C05442=1046.873,-51.756,-73.324,169.845,33.120,156.255
C05443=1046.866,-52.006,-73.312,169.843,33.118,156.255
C05444=1046.860,-52.255,-73.300,169.841,33.117,156.255
C05445=1046.854,-52.505,-73.288,169.839,33.117,156.255
C05446=1046.847,-52.754,-73.275,169.836,33.115,156.255
C05447=1046.841,-53.004,-73.262,169.834,33.114,156.255
C05448=1046.834,-53.254,-73.250,169.832,33.113,156.255
C05449=1046.828,-53.504,-73.238,169.830,33.112,156.255
C05450=1046.822,-53.753,-73.226,169.828,33.111,156.254
C05451=1046.815,-54.003,-73.214,169.826,33.110,156.254
C05452=1046.809,-54.253,-73.201,169.824,33.109,156.254
C05453=1046.802,-54.502,-73.189,169.822,33.108,156.254
C05454=1046.797,-54.752,-73.177,169.820,33.107,156.254
C05455=1046.790,-55.001,-73.165,169.817,33.106,156.254
C05456=1046.784,-55.251,-73.153,169.815,33.105,156.254
C05457=1046.778,-55.500,-73.140,169.813,33.104,156.254
C05458=1046.771,-55.749,-73.128,169.812,33.103,156.254
C05459=1046.764,-55.999,-73.116,169.810,33.102,156.253
C05460=1046.758,-56.249,-73.103,169.808,33.101,156.253
C05461=1046.752,-56.498,-73.092,169.806,33.100,156.253
C05462=1046.746,-56.748,-73.079,169.804,33.099,156.253
C05463=1046.739,-56.998,-73.067,169.801,33.098,156.253
C05464=1046.733,-57.247,-73.055,169.799,33.097,156.253
C05465=1046.727,-57.497,-73.043,169.797,33.096,156.253
C05466=1046.720,-57.747,-73.031,169.795,33.095,156.253
C05467=1046.714,-57.996,-73.019,169.793,33.094,156.253
C05468=1046.708,-58.246,-73.006,169.791,33.093,156.253
C05469=1046.701,-58.495,-72.994,169.789,33.092,156.253
C05470=1046.696,-58.746,-72.983,169.787,33.091,156.252
C05471=1046.689,-58.995,-72.971,169.784,33.090,156.252
C05472=1046.683,-59.245,-72.959,169.782,33.089,156.252
C05473=1046.677,-59.495,-72.946,169.780,33.088,156.252
C05474=1046.671,-59.744,-72.935,169.778,33.088,156.252
C05475=1046.664,-59.993,-72.923,169.776,33.086,156.252
C05476=1046.658,-60.243,-72.910,169.774,33.085,156.252
C05477=1046.651,-60.493,-72.898,169.772,33.085,156.252
C05478=1046.645,-60.742,-72.886,169.769,33.084,156.252
C05479=1046.639,-60.992,-72.874,169.767,33.082,156.252
C05480=1046.633,-61.242,-72.863,169.765,33.081,156.252
C05481=1046.626,-61.491,-72.851,169.763,33.081,156.251
C05482=1046.621,-61.741,-72.838,169.761,33.080,156.251
C05483=1046.614,-61.991,-72.826,169.759,33.079,156.251
C05484=1046.607,-62.240,-72.814,169.757,33.078,156.251
C05485=1046.602,-62.489,-72.802,169.755,33.077,156.251
C05486=1046.596,-62.740,-72.791,169.752,33.076,156.251
C05487=1046.589,-62.989,-72.779,169.750,33.075,156.251
C05488=1046.583,-63.239,-72.766,169.748,33.074,156.251
C05489=1046.576,-63.489,-72.754,169.746,33.073,156.251
C05490=1046.570,-63.737,-72.743,169.744,33.072,156.251
C05491=1046.565,-63.988,-72.731,169.742,33.071,156.251
C05492=1046.558,-64.238,-72.719,169.739,33.070,156.250
C05493=1046.551,-64.487,-72.707,169.738,33.069,156.250
C05494=1046.545,-64.736,-72.695,169.736,33.068,156.250
C05495=1046.540,-64.986,-72.684,169.734,33.067,156.250
C05496=1046.533,-65.236,-72.672,169.732,33.066,156.250
C05497=1046.527,-65.485,-72.660,169.730,33.065,156.250
C05498=1046.521,-65.735,-72.647,169.728,33.065,156.250
C05499=1046.515,-65.985,-72.636,169.725,33.064,156.250
C05500=1046.508,-66.235,-72.624,169.723,33.062,156.250
C05501=1046.503,-66.484,-72.612,169.721,33.061,156.250
C05502=1046.497,-66.734,-72.601,169.719,33.061,156.250
C05503=1046.489,-67.016,-72.587,169.716,33.060,156.250
C05504=1046.483,-67.299,-72.574,169.714,33.058,156.249
C05505=1046.476,-67.581,-72.560,169.712,33.057,156.249
C05506=1046.469,-67.863,-72.547,169.709,33.057,156.249
C05507=1046.462,-68.113,-72.535,169.707,33.056,156.249
C05508=1046.456,-68.362,-72.524,169.705,33.055,156.249
C05509=1046.450,-68.612,-72.513,169.703,33.054,156.249
C05510=1046.444,-68.862,-72.500,169.701,33.053,156.249
C05511=1046.438,-69.111,-72.489,169.698,33.052,156.249
C05512=1046.432,-69.361,-72.477,169.696,33.051,156.249
C05513=1046.425,-69.611,-72.465,169.694,33.050,156.249
C05514=1046.420,-69.860,-72.454,169.692,33.049,156.249
C05515=1046.413,-70.110,-72.442,169.690,33.049,156.248
C05516=1046.407,-70.360,-72.431,169.688,33.048,156.248
C05517=1046.401,-70.609,-72.419,169.685,33.047,156.248
C05518=1046.395,-70.859,-72.407,169.683,33.046,156.248
C05519=1046.389,-71.108,-72.396,169.681,33.045,156.248
C05520=1046.383,-71.358,-72.384,169.679,33.044,156.248
C05521=1046.376,-71.608,-72.372,169.677,33.043,156.248
C05522=1046.371,-71.857,-72.360,169.674,33.042,156.248
C05523=1046.365,-72.107,-72.349,169.672,33.041,156.248
C05524=1046.359,-72.356,-72.337,169.670,33.040,156.248
C05525=1046.352,-72.607,-72.326,169.669,33.040,156.248
C05526=1046.347,-72.856,-72.314,169.667,33.039,156.248
C05527=1046.341,-73.106,-72.303,169.665,33.038,156.248
C05528=1046.334,-73.356,-72.291,169.662,33.037,156.248
C05529=1046.328,-73.605,-72.280,169.660,33.036,156.247
C05530=1046.322,-73.855,-72.269,169.658,33.035,156.247
C05531=1046.317,-74.104,-72.256,169.656,33.035,156.247
C05532=1046.310,-74.355,-72.245,169.654,33.034,156.247
C05533=1046.304,-74.603,-72.234,169.651,33.033,156.247
C05534=1046.298,-74.854,-72.222,169.649,33.032,156.247
C05535=1046.292,-75.104,-72.211,169.647,33.031,156.247
C05536=1046.285,-75.352,-72.200,169.645,33.030,156.247
C05537=1046.278,-75.603,-72.189,169.643,33.030,156.247
C05538=1046.273,-75.852,-72.178,169.640,33.029,156.247
C05539=1046.266,-76.102,-72.166,169.638,33.028,156.247
C05540=1046.260,-76.351,-72.155,169.636,33.028,156.247
C05541=1046.254,-76.601,-72.144,169.634,33.027,156.247
C05542=1046.248,-76.850,-72.132,169.632,33.026,156.247
C05543=1046.242,-77.100,-72.121,169.629,33.025,156.247
C05544=1046.235,-77.351,-72.110,169.627,33.024,156.247
C05545=1046.229,-77.599,-72.098,169.625,33.024,156.247
C05546=1046.223,-77.850,-72.087,169.623,33.023,156.247
C05547=1046.217,-78.099,-72.076,169.620,33.022,156.247
C05548=1046.210,-78.349,-72.064,169.618,33.021,156.246
C05549=1046.205,-78.598,-72.053,169.616,33.021,156.246
C05550=1046.198,-78.848,-72.042,169.614,33.020,156.246
C05551=1046.193,-79.098,-72.031,169.612,33.020,156.246
C05552=1046.186,-79.348,-72.020,169.609,33.019,156.246
C05553=1046.180,-79.597,-72.008,169.607,33.018,156.246
C05554=1046.174,-79.847,-71.997,169.605,33.017,156.246
C05555=1046.167,-80.096,-71.987,169.603,33.016,156.246
C05556=1046.161,-80.346,-71.975,169.601,33.016,156.246
C05557=1046.155,-80.596,-71.965,169.599,33.015,156.246
C05558=1046.149,-80.846,-71.953,169.597,33.014,156.246
C05559=1046.142,-81.095,-71.942,169.595,33.014,156.246
C05560=1046.136,-81.345,-71.931,169.592,33.013,156.246
C05561=1046.130,-81.594,-71.920,169.590,33.012,156.246
C05562=1046.124,-81.845,-71.909,169.588,33.012,156.246
C05563=1046.117,-82.094,-71.899,169.586,33.011,156.246
C05564=1046.111,-82.344,-71.887,169.583,33.011,156.246
C05565=1046.105,-82.593,-71.877,169.581,33.010,156.246
C05566=1046.098,-82.843,-71.866,169.579,33.009,156.246
C05567=1046.091,-83.127,-71.853,169.576,33.009,156.246
C05568=1046.084,-83.412,-71.840,169.574,33.008,156.246
C05569=1046.077,-83.697,-71.828,169.571,33.007,156.246
C05570=1046.070,-83.981,-71.816,169.569,33.007,156.246
C05571=1046.063,-84.231,-71.804,169.566,33.006,156.246
C05572=1046.058,-84.480,-71.794,169.564,33.006,156.246
C05573=1046.051,-84.730,-71.783,169.562,33.005,156.246
C05574=1046.045,-84.980,-71.772,169.560,33.005,156.246
C05575=1046.039,-85.229,-71.761,169.557,33.004,156.246
C05576=1046.032,-85.479,-71.751,169.555,33.003,156.246
C05577=1046.026,-85.729,-71.740,169.553,33.003,156.246
C05578=1046.020,-85.979,-71.728,169.551,33.002,156.246
C05579=1046.013,-86.228,-71.718,169.548,33.002,156.246
C05580=1046.008,-86.477,-71.707,169.546,33.001,156.246
C05581=1046.001,-86.728,-71.696,169.544,33.000,156.246
C05582=1045.995,-86.977,-71.686,169.542,33.000,156.246
C05583=1045.989,-87.227,-71.674,169.540,32.999,156.246
C05584=1045.983,-87.477,-71.664,169.538,32.999,156.245
C05585=1045.977,-87.726,-71.654,169.536,32.998,156.246
C05586=1045.970,-87.977,-71.643,169.533,32.997,156.245
C05587=1045.965,-88.226,-71.632,169.531,32.997,156.246
C05588=1045.958,-88.475,-71.622,169.529,32.996,156.245
C05589=1045.952,-88.725,-71.610,169.527,32.996,156.246
C05590=1045.946,-88.975,-71.600,169.524,32.995,156.245
C05591=1045.940,-89.224,-71.589,169.522,32.995,156.245
C05592=1045.933,-89.474,-71.578,169.520,32.994,156.245
C05593=1045.927,-89.724,-71.567,169.518,32.994,156.245
C05594=1045.921,-89.974,-71.558,169.515,32.993,156.245
C05595=1045.915,-90.224,-71.546,169.513,32.993,156.245
C05596=1045.909,-90.473,-71.535,169.511,32.992,156.245
C05597=1045.903,-90.722,-71.525,169.508,32.992,156.245
C05598=1045.896,-90.973,-71.514,169.506,32.991,156.245
C05599=1045.890,-91.222,-71.504,169.504,32.991,156.245
C05600=1045.884,-91.472,-71.493,169.502,32.990,156.245
C05601=1045.878,-91.722,-71.482,169.499,32.990,156.245
C05602=1045.872,-91.971,-71.472,169.497,32.989,156.245
C05603=1045.866,-92.221,-71.461,169.495,32.989,156.245
C05604=1045.860,-92.470,-71.450,169.493,32.988,156.245
C05605=1045.853,-92.721,-71.440,169.490,32.988,156.245
C05606=1045.848,-92.970,-71.429,169.488,32.987,156.245
C05607=1045.841,-93.219,-71.419,169.486,32.987,156.245
C05608=1045.835,-93.469,-71.408,169.483,32.986,156.245
C05609=1045.829,-93.720,-71.398,169.481,32.986,156.245
C05610=1045.823,-93.969,-71.387,169.479,32.985,156.245
C05611=1045.817,-94.218,-71.377,169.477,32.985,156.245
C05612=1045.811,-94.468,-71.367,169.475,32.984,156.245
C05613=1045.805,-94.718,-71.356,169.473,32.983,156.245
C05614=1045.799,-94.968,-71.345,169.471,32.983,156.245
C05615=1045.792,-95.217,-71.335,169.468,32.982,156.245
C05616=1045.787,-95.467,-71.324,169.466,32.982,156.245
C05617=1045.781,-95.716,-71.314,169.464,32.982,156.245
C05618=1045.775,-95.966,-71.303,169.462,32.981,156.245
C05619=1045.769,-96.217,-71.293,169.459,32.981,156.245
C05620=1045.762,-96.466,-71.282,169.457,32.980,156.245
C05621=1045.757,-96.716,-71.272,169.455,32.980,156.245
C05622=1045.750,-96.965,-71.262,169.452,32.980,156.245
C05623=1045.745,-97.215,-71.251,169.450,32.979,156.245
C05624=1045.738,-97.465,-71.241,169.448,32.979,156.245
C05625=1045.732,-97.715,-71.230,169.446,32.978,156.245
C05626=1045.726,-97.964,-71.221,169.443,32.977,156.245
C05627=1045.720,-98.214,-71.210,169.441,32.977,156.245
C05628=1045.714,-98.463,-71.200,169.439,32.977,156.246
C05629=1045.707,-98.714,-71.190,169.436,32.977,156.246
C05630=1045.701,-98.963,-71.179,169.434,32.977,156.246
C05631=1045.695,-99.250,-71.168,169.431,32.976,156.246
C05632=1045.687,-99.536,-71.156,169.429,32.975,156.246
C05633=1045.680,-99.824,-71.145,169.426,32.975,156.246
C05634=1045.673,-100.111,-71.132,169.423,32.975,156.246
C05635=1045.667,-100.360,-71.123,169.421,32.974,156.246
C05636=1045.660,-100.610,-71.112,169.419,32.974,156.246
C05637=1045.655,-100.860,-71.102,169.416,32.974,156.246
C05638=1045.648,-101.109,-71.092,169.415,32.973,156.246
C05639=1045.642,-101.359,-71.082,169.413,32.973,156.246
C05640=1045.636,-101.608,-71.071,169.410,32.973,156.246
C05641=1045.629,-101.859,-71.061,169.408,32.972,156.246
C05642=1045.623,-102.108,-71.051,169.406,32.972,156.246
C05643=1045.618,-102.358,-71.041,169.403,32.972,156.246
C05644=1045.611,-102.608,-71.031,169.401,32.971,156.246
C05645=1045.605,-102.857,-71.021,169.399,32.971,156.246
C05646=1045.600,-103.107,-71.011,169.397,32.971,156.246
C05647=1045.593,-103.356,-71.001,169.394,32.971,156.246
C05648=1045.587,-103.606,-70.991,169.392,32.970,156.246
C05649=1045.581,-103.856,-70.982,169.390,32.970,156.246
C05650=1045.575,-104.105,-70.971,169.387,32.969,156.246
C05651=1045.569,-104.355,-70.961,169.385,32.969,156.246
C05652=1045.562,-104.606,-70.951,169.383,32.969,156.246
C05653=1045.556,-104.855,-70.940,169.380,32.969,156.246
C05654=1045.550,-105.105,-70.931,169.378,32.969,156.246
C05655=1045.544,-105.355,-70.921,169.376,32.968,156.246
C05656=1045.537,-105.604,-70.911,169.373,32.968,156.246
C05657=1045.532,-105.854,-70.901,169.371,32.968,156.247
C05658=1045.526,-106.104,-70.891,169.369,32.968,156.247
C05659=1045.520,-106.354,-70.882,169.366,32.967,156.247
C05660=1045.513,-106.603,-70.871,169.364,32.967,156.247
C05661=1045.507,-106.853,-70.862,169.362,32.966,156.247
C05662=1045.502,-107.103,-70.852,169.359,32.966,156.247
C05663=1045.495,-107.352,-70.842,169.357,32.966,156.247
C05664=1045.489,-107.602,-70.832,169.355,32.966,156.247
C05665=1045.483,-107.851,-70.822,169.353,32.966,156.247
C05666=1045.477,-108.101,-70.813,169.351,32.965,156.247
C05667=1045.470,-108.351,-70.803,169.349,32.966,156.247
C05668=1045.465,-108.601,-70.792,169.346,32.965,156.247
C05669=1045.459,-108.850,-70.783,169.344,32.965,156.247
C05670=1045.452,-109.100,-70.773,169.341,32.965,156.247
C05671=1045.446,-109.350,-70.763,169.339,32.965,156.247
C05672=1045.440,-109.600,-70.754,169.337,32.965,156.247
C05673=1045.434,-109.850,-70.744,169.334,32.964,156.247
C05674=1045.427,-110.099,-70.734,169.332,32.964,156.247
C05675=1045.421,-110.348,-70.725,169.330,32.964,156.247
C05676=1045.415,-110.598,-70.715,169.327,32.964,156.247
C05677=1045.409,-110.848,-70.705,169.325,32.963,156.248
C05678=1045.403,-111.098,-70.695,169.323,32.964,156.248
C05679=1045.397,-111.348,-70.686,169.320,32.964,156.248
C05680=1045.391,-111.598,-70.676,169.318,32.963,156.248
C05681=1045.385,-111.848,-70.667,169.316,32.963,156.248
C05682=1045.379,-112.097,-70.657,169.313,32.963,156.248
C05683=1045.373,-112.347,-70.647,169.311,32.963,156.248
C05684=1045.366,-112.597,-70.638,169.308,32.962,156.248
C05685=1045.360,-112.846,-70.628,169.306,32.962,156.248
C05686=1045.354,-113.096,-70.618,169.304,32.963,156.248
C05687=1045.348,-113.346,-70.608,169.301,32.962,156.248
C05688=1045.342,-113.595,-70.599,169.299,32.962,156.248
C05689=1045.336,-113.845,-70.590,169.297,32.962,156.248
C05690=1045.330,-114.094,-70.580,169.295,32.962,156.248
C05691=1045.323,-114.344,-70.570,169.293,32.962,156.248
C05692=1045.317,-114.594,-70.561,169.291,32.962,156.249
C05693=1045.311,-114.844,-70.551,169.288,32.962,156.249
C05694=1045.305,-115.094,-70.542,169.286,32.962,156.249
C05695=1045.298,-115.380,-70.531,169.283,32.961,156.249
C05696=1045.291,-115.665,-70.520,169.280,32.962,156.249
C05697=1045.284,-115.952,-70.509,169.278,32.961,156.249
C05698=1045.277,-116.237,-70.499,169.275,32.961,156.249
C05699=1045.271,-116.487,-70.489,169.273,32.962,156.249
C05700=1045.265,-116.736,-70.480,169.270,32.961,156.249
C05701=1045.259,-116.986,-70.470,169.268,32.961,156.249
C05702=1045.253,-117.237,-70.461,169.266,32.962,156.249
C05703=1045.247,-117.486,-70.452,169.263,32.961,156.250
C05704=1045.240,-117.736,-70.442,169.261,32.961,156.250
C05705=1045.235,-117.985,-70.433,169.258,32.961,156.250
C05706=1045.229,-118.235,-70.423,169.256,32.961,156.250
C05707=1045.223,-118.485,-70.414,169.254,32.961,156.250
C05708=1045.216,-118.734,-70.405,169.251,32.961,156.250
C05709=1045.210,-118.985,-70.396,169.249,32.961,156.250
C05710=1045.204,-119.235,-70.386,169.247,32.961,156.250
C05711=1045.198,-119.484,-70.377,169.244,32.961,156.250
C05712=1045.192,-119.733,-70.368,169.242,32.961,156.250
C05713=1045.186,-119.983,-70.358,169.239,32.961,156.250
C05714=1045.180,-120.234,-70.349,169.237,32.961,156.251
C05715=1045.174,-120.483,-70.340,169.235,32.961,156.251
C05716=1045.167,-120.732,-70.331,169.233,32.961,156.251
C05717=1045.161,-120.982,-70.321,169.231,32.961,156.251
C05718=1045.155,-121.232,-70.312,169.228,32.961,156.251
C05719=1045.149,-121.482,-70.303,169.226,32.962,156.251
C05720=1045.143,-121.732,-70.293,169.224,32.961,156.251
C05721=1045.137,-121.981,-70.284,169.221,32.962,156.251
C05722=1045.130,-122.231,-70.275,169.219,32.961,156.251
C05723=1045.125,-122.481,-70.266,169.217,32.961,156.251
C05724=1045.118,-122.731,-70.257,169.214,32.962,156.251
C05725=1045.113,-122.980,-70.248,169.212,32.961,156.252
C05726=1045.107,-123.230,-70.239,169.209,32.962,156.252
C05727=1045.101,-123.480,-70.229,169.207,32.962,156.252
C05728=1045.094,-123.730,-70.220,169.205,32.962,156.252
C05729=1045.089,-123.979,-70.212,169.202,32.962,156.252
C05730=1045.083,-124.229,-70.202,169.200,32.962,156.252
C05731=1045.076,-124.479,-70.193,169.197,32.962,156.252
C05732=1045.070,-124.729,-70.184,169.195,32.962,156.252
C05733=1045.064,-124.978,-70.175,169.193,32.962,156.252
C05734=1045.058,-125.228,-70.166,169.190,32.963,156.253
C05735=1045.052,-125.478,-70.157,169.188,32.962,156.253
C05736=1045.045,-125.728,-70.148,169.185,32.963,156.253
C05737=1045.040,-125.978,-70.139,169.183,32.963,156.253
C05738=1045.034,-126.227,-70.130,169.181,32.963,156.253
C05739=1045.027,-126.478,-70.122,169.178,32.963,156.253
C05740=1045.022,-126.727,-70.112,169.176,32.963,156.253
C05741=1045.015,-126.976,-70.103,169.174,32.964,156.253
C05742=1045.009,-127.227,-70.094,169.172,32.964,156.254
C05743=1045.003,-127.476,-70.085,169.170,32.964,156.254
C05744=1044.997,-127.726,-70.076,169.167,32.964,156.254
C05745=1044.992,-127.975,-70.067,169.165,32.964,156.254
C05746=1044.986,-128.225,-70.057,169.163,32.963,156.254
C05747=1044.982,-128.475,-70.047,169.161,32.962,156.254
C05748=1044.980,-128.725,-70.035,169.159,32.961,156.253
C05749=1044.978,-128.975,-70.024,169.157,32.959,156.253
C05750=1044.977,-129.225,-70.011,169.155,32.957,156.253
C05751=1044.977,-129.475,-69.999,169.153,32.954,156.252
C05752=1044.978,-129.725,-69.985,169.152,32.951,156.252
C05753=1044.979,-129.976,-69.971,169.150,32.947,156.251
C05754=1044.982,-130.225,-69.957,169.149,32.943,156.251
C05755=1044.986,-130.476,-69.941,169.148,32.938,156.250
C05756=1044.990,-130.727,-69.925,169.147,32.933,156.249
C05757=1044.995,-130.977,-69.908,169.146,32.927,156.248
C05758=1045.002,-131.227,-69.891,169.145,32.921,156.247
C05759=1044.646,-131.251,-70.134,169.099,33.102,156.280
C05760=1044.641,-131.000,-70.151,169.100,33.108,156.281
C05761=1044.635,-130.751,-70.168,169.101,33.114,156.282
C05762=1044.631,-130.500,-70.184,169.102,33.119,156.283
C05763=1044.627,-130.249,-70.199,169.103,33.124,156.283
C05764=1044.624,-129.999,-70.214,169.104,33.128,156.284
C05765=1044.622,-129.749,-70.229,169.105,33.131,156.285
C05766=1044.622,-129.499,-70.242,169.107,33.135,156.285
C05767=1044.622,-129.248,-70.255,169.108,33.138,156.285
C05768=1044.623,-128.998,-70.268,169.110,33.140,156.286
C05769=1044.625,-128.749,-70.279,169.112,33.142,156.286
C05770=1044.627,-128.498,-70.291,169.114,33.144,156.286
C05771=1044.631,-128.249,-70.301,169.116,33.145,156.286
C05772=1044.636,-127.999,-70.311,169.118,33.145,156.286
C05773=1044.641,-127.749,-70.320,169.121,33.145,156.286
C05774=1044.648,-127.500,-70.329,169.123,33.145,156.286
C05775=1044.653,-127.251,-70.338,169.125,33.145,156.286
C05776=1044.659,-127.000,-70.347,169.128,33.144,156.286
C05777=1044.666,-126.751,-70.356,169.130,33.145,156.286
C05778=1044.671,-126.501,-70.364,169.133,33.144,156.286
C05779=1044.677,-126.251,-70.374,169.135,33.144,156.286
C05780=1044.684,-126.001,-70.382,169.138,33.144,156.285
C05781=1044.690,-125.751,-70.392,169.140,33.144,156.285
C05782=1044.696,-125.502,-70.400,169.142,33.144,156.285
C05783=1044.702,-125.252,-70.409,169.145,33.143,156.285
C05784=1044.709,-125.002,-70.419,169.147,33.143,156.285
C05785=1044.714,-124.753,-70.427,169.149,33.143,156.285
C05786=1044.721,-124.503,-70.436,169.151,33.143,156.285
C05787=1044.727,-124.253,-70.446,169.153,33.143,156.285
C05788=1044.733,-124.003,-70.455,169.156,33.143,156.285
C05789=1044.738,-123.754,-70.464,169.158,33.143,156.285
C05790=1044.745,-123.504,-70.473,169.161,33.142,156.284
C05791=1044.751,-123.254,-70.482,169.163,33.143,156.284
C05792=1044.757,-123.004,-70.491,169.165,33.142,156.284
C05793=1044.763,-122.755,-70.500,169.168,33.142,156.284
C05794=1044.769,-122.505,-70.509,169.170,33.142,156.284
C05795=1044.775,-122.255,-70.519,169.173,33.142,156.284
C05796=1044.782,-122.005,-70.528,169.175,33.142,156.284
C05797=1044.787,-121.756,-70.536,169.177,33.142,156.284
C05798=1044.793,-121.506,-70.546,169.180,33.142,156.284
C05799=1044.799,-121.256,-70.555,169.182,33.142,156.283
C05800=1044.806,-121.006,-70.565,169.185,33.142,156.283
C05801=1044.812,-120.756,-70.574,169.187,33.142,156.283
C05802=1044.817,-120.507,-70.583,169.189,33.142,156.283
C05803=1044.824,-120.257,-70.592,169.192,33.141,156.283
C05804=1044.830,-120.008,-70.602,169.194,33.142,156.283
C05805=1044.836,-119.758,-70.611,169.197,33.141,156.283
C05806=1044.842,-119.507,-70.620,169.199,33.141,156.283
C05807=1044.848,-119.258,-70.629,169.201,33.142,156.283
C05808=1044.854,-119.008,-70.639,169.204,33.141,156.283
C05809=1044.860,-118.759,-70.648,169.206,33.141,156.283
C05810=1044.866,-118.509,-70.658,169.208,33.142,156.282
C05811=1044.873,-118.259,-70.667,169.210,33.141,156.282
C05812=1044.879,-118.009,-70.676,169.212,33.141,156.282
C05813=1044.885,-117.760,-70.685,169.215,33.141,156.282
C05814=1044.891,-117.510,-70.694,169.217,33.141,156.282
C05815=1044.897,-117.260,-70.704,169.220,33.141,156.282
C05816=1044.903,-117.010,-70.714,169.222,33.141,156.282
C05817=1044.909,-116.761,-70.723,169.224,33.141,156.282
C05818=1044.915,-116.511,-70.733,169.227,33.141,156.282
C05819=1044.922,-116.261,-70.742,169.229,33.141,156.282
C05820=1044.929,-115.975,-70.752,169.232,33.141,156.282
C05821=1044.936,-115.689,-70.764,169.235,33.141,156.281
C05822=1044.943,-115.403,-70.774,169.237,33.141,156.281
C05823=1044.949,-115.118,-70.785,169.240,33.141,156.281
C05824=1044.956,-114.868,-70.795,169.242,33.141,156.281
C05825=1044.962,-114.618,-70.804,169.245,33.142,156.281
C05826=1044.968,-114.369,-70.814,169.247,33.141,156.281
C05827=1044.974,-114.119,-70.824,169.249,33.141,156.281
C05828=1044.980,-113.869,-70.833,169.252,33.142,156.281
C05829=1044.986,-113.619,-70.843,169.254,33.142,156.281
C05830=1044.992,-113.370,-70.852,169.257,33.142,156.281
C05831=1044.998,-113.120,-70.861,169.259,33.142,156.281
C05832=1045.004,-112.870,-70.871,169.261,33.142,156.281
C05833=1045.011,-112.621,-70.881,169.264,33.142,156.281
C05834=1045.017,-112.371,-70.890,169.266,33.142,156.281
C05835=1045.023,-112.121,-70.900,169.268,33.143,156.280
C05836=1045.029,-111.871,-70.909,169.270,33.142,156.280
C05837=1045.035,-111.621,-70.919,169.272,33.142,156.280
C05838=1045.041,-111.371,-70.929,169.275,33.143,156.280
C05839=1045.047,-111.122,-70.939,169.277,33.143,156.280
C05840=1045.053,-110.872,-70.948,169.279,33.143,156.280
C05841=1045.059,-110.622,-70.958,169.282,33.143,156.280
C05842=1045.066,-110.373,-70.968,169.284,33.143,156.280
C05843=1045.072,-110.123,-70.978,169.286,33.143,156.280
C05844=1045.078,-109.873,-70.987,169.289,33.143,156.280
C05845=1045.084,-109.623,-70.997,169.291,33.143,156.280
C05846=1045.090,-109.374,-71.006,169.293,33.144,156.280
C05847=1045.096,-109.124,-71.016,169.296,33.144,156.280
C05848=1045.103,-108.874,-71.025,169.298,33.144,156.280
C05849=1045.108,-108.624,-71.036,169.301,33.144,156.280
C05850=1045.115,-108.375,-71.046,169.303,33.145,156.280
C05851=1045.121,-108.125,-71.055,169.305,33.145,156.280
C05852=1045.127,-107.875,-71.065,169.308,33.144,156.279
C05853=1045.133,-107.625,-71.075,169.310,33.144,156.279
C05854=1045.140,-107.376,-71.085,169.312,33.145,156.279
C05855=1045.146,-107.126,-71.094,169.315,33.145,156.279
C05856=1045.151,-106.876,-71.105,169.317,33.145,156.279
C05857=1045.157,-106.626,-71.114,169.319,33.145,156.279
C05858=1045.164,-106.377,-71.124,169.322,33.146,156.279
C05859=1045.170,-106.127,-71.134,169.324,33.146,156.279
C05860=1045.175,-105.877,-71.144,169.326,33.146,156.279
C05861=1045.182,-105.628,-71.154,169.329,33.146,156.279
C05862=1045.188,-105.378,-71.164,169.331,33.146,156.279
C05863=1045.194,-105.129,-71.174,169.333,33.147,156.279
C05864=1045.200,-104.878,-71.184,169.335,33.147,156.279
C05865=1045.206,-104.629,-71.194,169.337,33.148,156.279
C05866=1045.212,-104.379,-71.204,169.339,33.148,156.279
C05867=1045.219,-104.129,-71.213,169.342,33.148,156.279
C05868=1045.225,-103.879,-71.224,169.344,33.148,156.279
C05869=1045.231,-103.630,-71.234,169.346,33.148,156.279
C05870=1045.237,-103.380,-71.244,169.349,33.149,156.279
C05871=1045.243,-103.130,-71.254,169.351,33.149,156.279
C05872=1045.249,-102.881,-71.264,169.353,33.149,156.279
C05873=1045.256,-102.631,-71.274,169.356,33.149,156.278
C05874=1045.262,-102.382,-71.284,169.358,33.150,156.278
C05875=1045.267,-102.132,-71.295,169.360,33.150,156.278
C05876=1045.274,-101.882,-71.304,169.363,33.151,156.278
C05877=1045.280,-101.632,-71.314,169.365,33.151,156.278
C05878=1045.286,-101.382,-71.325,169.367,33.151,156.278
C05879=1045.292,-101.133,-71.335,169.370,33.151,156.278
C05880=1045.299,-100.883,-71.345,169.372,33.151,156.278
C05881=1045.304,-100.633,-71.355,169.374,33.152,156.278
C05882=1045.311,-100.384,-71.365,169.377,33.152,156.278
C05883=1045.317,-100.134,-71.375,169.379,33.153,156.278
C05884=1045.324,-99.847,-71.387,169.382,33.153,156.278
C05885=1045.331,-99.560,-71.399,169.384,33.153,156.278
C05886=1045.339,-99.273,-71.411,169.387,33.153,156.278
C05887=1045.345,-98.986,-71.422,169.390,33.154,156.278
C05888=1045.351,-98.737,-71.432,169.392,33.155,156.278
C05889=1045.358,-98.487,-71.442,169.394,33.155,156.278
C05890=1045.364,-98.237,-71.453,169.397,33.155,156.278
C05891=1045.370,-97.987,-71.463,169.399,33.155,156.278
C05892=1045.376,-97.738,-71.473,169.400,33.155,156.278
C05893=1045.382,-97.489,-71.484,169.403,33.156,156.278
C05894=1045.389,-97.238,-71.494,169.405,33.156,156.278
C05895=1045.395,-96.989,-71.505,169.407,33.157,156.278
C05896=1045.401,-96.739,-71.514,169.410,33.158,156.278
C05897=1045.406,-96.489,-71.525,169.412,33.158,156.278
C05898=1045.412,-96.240,-71.536,169.414,33.158,156.278
C05899=1045.418,-95.990,-71.546,169.417,33.159,156.278
C05900=1045.425,-95.740,-71.557,169.419,33.159,156.278
C05901=1045.431,-95.491,-71.567,169.421,33.159,156.278
C05902=1045.437,-95.241,-71.577,169.423,33.160,156.278
C05903=1045.443,-94.991,-71.588,169.426,33.160,156.278
C05904=1045.449,-94.742,-71.598,169.428,33.161,156.278
C05905=1045.455,-94.491,-71.609,169.430,33.161,156.278
C05906=1045.461,-94.242,-71.619,169.433,33.161,156.278
C05907=1045.467,-93.992,-71.630,169.435,33.162,156.278
C05908=1045.474,-93.743,-71.640,169.437,33.162,156.278
C05909=1045.480,-93.493,-71.651,169.439,33.163,156.278
C05910=1045.485,-93.243,-71.662,169.442,33.164,156.278
C05911=1045.492,-92.994,-71.672,169.444,33.164,156.278
C05912=1045.498,-92.744,-71.683,169.446,33.165,156.278
C05913=1045.504,-92.494,-71.693,169.449,33.165,156.278
C05914=1045.510,-92.244,-71.704,169.451,33.166,156.278
C05915=1045.516,-91.995,-71.715,169.453,33.166,156.278
C05916=1045.522,-91.746,-71.725,169.456,33.167,156.278
C05917=1045.528,-91.495,-71.736,169.458,33.167,156.278
C05918=1045.534,-91.245,-71.746,169.460,33.167,156.278
C05919=1045.541,-90.996,-71.757,169.462,33.168,156.278
C05920=1045.547,-90.746,-71.768,169.465,33.168,156.278
C05921=1045.553,-90.497,-71.778,169.467,33.169,156.278
C05922=1045.559,-90.247,-71.789,169.468,33.169,156.278
C05923=1045.565,-89.997,-71.799,169.470,33.170,156.278
C05924=1045.572,-89.747,-71.810,169.473,33.170,156.278
C05925=1045.577,-89.498,-71.821,169.475,33.171,156.278
C05926=1045.583,-89.248,-71.832,169.477,33.171,156.278
C05927=1045.590,-88.999,-71.842,169.480,33.172,156.278
C05928=1045.596,-88.749,-71.853,169.482,33.172,156.278
C05929=1045.602,-88.500,-71.864,169.484,33.173,156.278
C05930=1045.609,-88.250,-71.875,169.486,33.173,156.278
C05931=1045.614,-88.000,-71.885,169.489,33.174,156.278
C05932=1045.621,-87.749,-71.896,169.491,33.174,156.278
C05933=1045.627,-87.500,-71.906,169.493,33.175,156.278
C05934=1045.633,-87.251,-71.917,169.496,33.175,156.278
C05935=1045.639,-87.000,-71.928,169.498,33.176,156.278
C05936=1045.646,-86.751,-71.939,169.500,33.176,156.278
C05937=1045.651,-86.502,-71.950,169.502,33.177,156.278
C05938=1045.658,-86.252,-71.961,169.505,33.178,156.278
C05939=1045.664,-86.002,-71.971,169.507,33.178,156.278
C05940=1045.670,-85.752,-71.982,169.509,33.179,156.278
C05941=1045.676,-85.503,-71.993,169.511,33.179,156.278
C05942=1045.683,-85.254,-72.004,169.514,33.180,156.278
C05943=1045.689,-85.003,-72.015,169.516,33.180,156.278
C05944=1045.695,-84.754,-72.026,169.518,33.181,156.278
C05945=1045.702,-84.504,-72.036,169.521,33.182,156.278
C05946=1045.708,-84.255,-72.047,169.523,33.182,156.278
C05947=1045.714,-84.004,-72.058,169.525,33.183,156.278
C05948=1045.721,-83.720,-72.071,169.528,33.183,156.278
C05949=1045.728,-83.436,-72.083,169.530,33.184,156.278
C05950=1045.735,-83.151,-72.096,169.533,33.185,156.278
C05951=1045.742,-82.866,-72.108,169.535,33.185,156.278
C05952=1045.749,-82.616,-72.119,169.538,33.186,156.278
C05953=1045.755,-82.367,-72.130,169.539,33.186,156.278
C05954=1045.761,-82.117,-72.141,169.541,33.187,156.278
C05955=1045.768,-81.868,-72.152,169.543,33.187,156.278
C05956=1045.774,-81.618,-72.163,169.546,33.188,156.278
C05957=1045.780,-81.369,-72.174,169.548,33.188,156.278
C05958=1045.786,-81.118,-72.185,169.550,33.189,156.278
C05959=1045.793,-80.869,-72.195,169.552,33.190,156.278
C05960=1045.799,-80.619,-72.207,169.555,33.190,156.278
C05961=1045.805,-80.369,-72.218,169.557,33.191,156.278
C05962=1045.812,-80.120,-72.230,169.559,33.192,156.279
C05963=1045.818,-79.871,-72.240,169.561,33.192,156.278
C05964=1045.824,-79.621,-72.251,169.564,33.193,156.279
C05965=1045.830,-79.371,-72.262,169.566,33.194,156.279
C05966=1045.836,-79.121,-72.273,169.568,33.194,156.279
C05967=1045.843,-78.872,-72.285,169.570,33.195,156.279
C05968=1045.849,-78.622,-72.296,169.573,33.196,156.279
C05969=1045.855,-78.372,-72.307,169.575,33.197,156.279
C05970=1045.861,-78.122,-72.318,169.577,33.197,156.279
C05971=1045.867,-77.873,-72.330,169.579,33.198,156.279
C05972=1045.873,-77.623,-72.341,169.582,33.198,156.279
C05973=1045.879,-77.374,-72.352,169.584,33.199,156.279
C05974=1045.886,-77.124,-72.364,169.586,33.200,156.279
C05975=1045.891,-76.874,-72.375,169.588,33.201,156.279
C05976=1045.898,-76.624,-72.386,169.590,33.202,156.279
C05977=1045.904,-76.374,-72.397,169.593,33.202,156.279
C05978=1045.910,-76.125,-72.409,169.595,33.203,156.279
C05979=1045.917,-75.875,-72.420,169.597,33.204,156.279
C05980=1045.923,-75.626,-72.432,169.599,33.204,156.279
C05981=1045.930,-75.376,-72.442,169.602,33.205,156.279
C05982=1045.935,-75.127,-72.453,169.604,33.206,156.279
C05983=1045.942,-74.877,-72.465,169.606,33.206,156.279
C05984=1045.948,-74.627,-72.476,169.608,33.207,156.279
C05985=1045.954,-74.378,-72.487,169.610,33.208,156.280
C05986=1045.961,-74.128,-72.499,169.613,33.209,156.280
C05987=1045.966,-73.878,-72.510,169.614,33.210,156.280
C05988=1045.972,-73.629,-72.523,169.616,33.210,156.280
C05989=1045.978,-73.379,-72.533,169.618,33.211,156.280
C05990=1045.985,-73.130,-72.545,169.620,33.212,156.280
C05991=1045.991,-72.879,-72.557,169.623,33.213,156.280
C05992=1045.996,-72.630,-72.569,169.625,33.214,156.280
C05993=1046.003,-72.380,-72.580,169.627,33.215,156.280
C05994=1046.009,-72.131,-72.592,169.629,33.215,156.280
C05995=1046.015,-71.881,-72.603,169.631,33.216,156.280
C05996=1046.020,-71.632,-72.615,169.633,33.217,156.280
C05997=1046.027,-71.382,-72.626,169.636,33.218,156.280
C05998=1046.033,-71.132,-72.638,169.638,33.219,156.280
C05999=1046.039,-70.882,-72.649,169.640,33.220,156.280
C06000=1046.045,-70.633,-72.662,169.642,33.220,156.281
C06001=1046.051,-70.383,-72.673,169.644,33.221,156.281
C06002=1046.057,-70.134,-72.685,169.647,33.222,156.281
C06003=1046.064,-69.883,-72.696,169.649,33.223,156.281
C06004=1046.069,-69.634,-72.708,169.651,33.224,156.281
C06005=1046.076,-69.385,-72.720,169.653,33.225,156.281
C06006=1046.082,-69.134,-72.731,169.655,33.226,156.281
C06007=1046.088,-68.886,-72.743,169.657,33.227,156.281
C06008=1046.094,-68.635,-72.755,169.660,33.228,156.281
C06009=1046.100,-68.386,-72.766,169.662,33.228,156.281
C06010=1046.106,-68.137,-72.778,169.664,33.229,156.281
C06011=1046.113,-67.886,-72.789,169.666,33.230,156.281
C06012=1046.120,-67.604,-72.803,169.669,33.231,156.281
C06013=1046.127,-67.322,-72.816,169.671,33.232,156.282
C06014=1046.134,-67.040,-72.830,169.673,33.233,156.282
C06015=1046.140,-66.757,-72.843,169.676,33.234,156.282
C06016=1046.147,-66.507,-72.855,169.678,33.235,156.282
C06017=1046.152,-66.258,-72.866,169.680,33.236,156.282
C06018=1046.159,-66.008,-72.878,169.682,33.237,156.282
C06019=1046.165,-65.758,-72.890,169.685,33.238,156.282
C06020=1046.171,-65.509,-72.903,169.687,33.239,156.282
C06021=1046.177,-65.259,-72.914,169.689,33.240,156.282
C06022=1046.184,-65.009,-72.926,169.691,33.240,156.282
C06023=1046.190,-64.760,-72.938,169.693,33.241,156.282
C06024=1046.196,-64.510,-72.950,169.695,33.242,156.282
C06025=1046.202,-64.261,-72.961,169.697,33.243,156.283
C06026=1046.209,-64.011,-72.973,169.699,33.244,156.283
C06027=1046.214,-63.761,-72.986,169.701,33.245,156.283
C06028=1046.221,-63.511,-72.997,169.703,33.246,156.283
C06029=1046.227,-63.262,-73.008,169.705,33.247,156.283
C06030=1046.233,-63.012,-73.021,169.707,33.248,156.283
C06031=1046.239,-62.763,-73.033,169.709,33.248,156.283
C06032=1046.246,-62.513,-73.045,169.712,33.250,156.283
C06033=1046.251,-62.264,-73.057,169.714,33.251,156.283
C06034=1046.258,-62.014,-73.069,169.716,33.252,156.283
C06035=1046.264,-61.764,-73.080,169.718,33.252,156.283
C06036=1046.270,-61.514,-73.093,169.720,33.253,156.284
C06037=1046.277,-61.265,-73.105,169.722,33.254,156.284
C06038=1046.283,-61.016,-73.116,169.725,33.255,156.284
C06039=1046.289,-60.766,-73.129,169.727,33.256,156.284
C06040=1046.296,-60.516,-73.141,169.729,33.257,156.284
C06041=1046.302,-60.267,-73.153,169.731,33.258,156.284
C06042=1046.308,-60.016,-73.165,169.733,33.259,156.284
C06043=1046.314,-59.767,-73.177,169.735,33.260,156.284
C06044=1046.320,-59.518,-73.188,169.737,33.261,156.284
C06045=1046.326,-59.268,-73.201,169.740,33.262,156.284
C06046=1046.333,-59.018,-73.213,169.742,33.263,156.284
C06047=1046.340,-58.769,-73.225,169.744,33.263,156.285
C06048=1046.346,-58.519,-73.237,169.746,33.265,156.285
C06049=1046.352,-58.269,-73.249,169.748,33.266,156.285
C06050=1046.359,-58.020,-73.261,169.750,33.266,156.285
C06051=1046.365,-57.770,-73.274,169.752,33.267,156.285
C06052=1046.371,-57.521,-73.285,169.755,33.268,156.285
C06053=1046.377,-57.271,-73.298,169.757,33.270,156.285
C06054=1046.383,-57.021,-73.310,169.759,33.270,156.285
C06055=1046.390,-56.772,-73.322,169.761,33.271,156.285
C06056=1046.396,-56.522,-73.334,169.763,33.272,156.285
C06057=1046.403,-56.272,-73.346,169.765,33.273,156.286
C06058=1046.409,-56.023,-73.358,169.767,33.274,156.286
C06059=1046.415,-55.773,-73.371,169.769,33.275,156.286
C06060=1046.422,-55.523,-73.383,169.772,33.276,156.286
C06061=1046.428,-55.274,-73.395,169.774,33.277,156.286
C06062=1046.434,-55.024,-73.407,169.776,33.278,156.286
C06063=1046.441,-54.774,-73.419,169.778,33.279,156.286
C06064=1046.447,-54.525,-73.432,169.780,33.280,156.286
C06065=1046.453,-54.276,-73.443,169.782,33.281,156.286
C06066=1046.459,-54.026,-73.456,169.784,33.282,156.286
C06067=1046.465,-53.776,-73.468,169.786,33.283,156.287
C06068=1046.472,-53.527,-73.481,169.789,33.284,156.287
C06069=1046.478,-53.277,-73.493,169.790,33.285,156.287
C06070=1046.485,-53.028,-73.505,169.792,33.286,156.287
C06071=1046.491,-52.778,-73.518,169.794,33.287,156.287
C06072=1046.498,-52.528,-73.530,169.796,33.288,156.287
C06073=1046.504,-52.279,-73.542,169.798,33.289,156.287
C06074=1046.510,-52.029,-73.554,169.800,33.290,156.287
C06075=1046.517,-51.780,-73.567,169.802,33.291,156.287
C06076=1046.524,-51.498,-73.580,169.805,33.292,156.287
C06077=1046.531,-51.217,-73.595,169.807,33.293,156.288
C06078=1046.539,-50.936,-73.608,169.810,33.294,156.288
C06079=1046.546,-50.655,-73.622,169.812,33.295,156.288
C06080=1046.552,-50.405,-73.635,169.814,33.296,156.288
C06081=1046.558,-50.156,-73.647,169.816,33.298,156.288
C06082=1046.564,-49.906,-73.659,169.818,33.298,156.288
C06083=1046.570,-49.657,-73.673,169.820,33.300,156.288
C06084=1046.576,-49.407,-73.685,169.822,33.301,156.288
C06085=1046.583,-49.157,-73.697,169.824,33.302,156.289
C06086=1046.589,-48.907,-73.710,169.826,33.303,156.289
C06087=1046.595,-48.658,-73.723,169.829,33.304,156.289
C06088=1046.601,-48.408,-73.736,169.831,33.306,156.289
C06089=1046.608,-48.159,-73.748,169.833,33.307,156.289
C06090=1046.614,-47.909,-73.761,169.835,33.308,156.289
C06091=1046.620,-47.660,-73.773,169.837,33.309,156.289
C06092=1046.626,-47.410,-73.787,169.839,33.310,156.290
C06093=1046.633,-47.161,-73.799,169.841,33.311,156.290
C06094=1046.639,-46.911,-73.811,169.843,33.312,156.290
C06095=1046.645,-46.661,-73.825,169.845,33.313,156.290
C06096=1046.651,-46.411,-73.837,169.847,33.315,156.290
C06097=1046.658,-46.161,-73.849,169.849,33.315,156.290
C06098=1046.664,-45.912,-73.863,169.851,33.317,156.290
C06099=1046.670,-45.662,-73.875,169.853,33.318,156.290
C06100=1046.676,-45.413,-73.888,169.855,33.319,156.291
C06101=1046.682,-45.163,-73.901,169.857,33.321,156.291
C06102=1046.689,-44.914,-73.913,169.859,33.321,156.291
C06103=1046.695,-44.664,-73.926,169.862,33.323,156.291
C06104=1046.701,-44.414,-73.939,169.864,33.324,156.291
C06105=1046.707,-44.165,-73.952,169.866,33.325,156.291
C06106=1046.713,-43.915,-73.965,169.868,33.326,156.291
C06107=1046.720,-43.666,-73.977,169.870,33.327,156.292
C06108=1046.726,-43.416,-73.990,169.872,33.329,156.292
C06109=1046.733,-43.166,-74.003,169.874,33.330,156.292
C06110=1046.739,-42.917,-74.016,169.876,33.331,156.292
C06111=1046.745,-42.667,-74.029,169.878,33.332,156.292
C06112=1046.751,-42.418,-74.041,169.880,33.333,156.292
C06113=1046.758,-42.168,-74.055,169.882,33.335,156.292
C06114=1046.764,-41.919,-74.067,169.884,33.335,156.292
C06115=1046.770,-41.669,-74.080,169.886,33.337,156.293
C06116=1046.776,-41.419,-74.093,169.888,33.338,156.293
C06117=1046.783,-41.170,-74.106,169.890,33.339,156.293
C06118=1046.789,-40.921,-74.119,169.892,33.340,156.293
C06119=1046.795,-40.671,-74.132,169.894,33.341,156.293
C06120=1046.802,-40.421,-74.145,169.896,33.343,156.293
C06121=1046.807,-40.171,-74.158,169.898,33.344,156.293
C06122=1046.814,-39.923,-74.170,169.900,33.345,156.294
C06123=1046.821,-39.672,-74.183,169.902,33.346,156.294
C06124=1046.827,-39.423,-74.196,169.904,33.347,156.294
C06125=1046.833,-39.173,-74.210,169.907,33.349,156.294
C06126=1046.839,-38.924,-74.222,169.909,33.349,156.294
C06127=1046.846,-38.674,-74.236,169.910,33.351,156.294
C06128=1046.852,-38.425,-74.249,169.912,33.352,156.295
C06129=1046.858,-38.174,-74.262,169.914,33.353,156.295
C06130=1046.864,-37.925,-74.275,169.916,33.355,156.295
C06131=1046.871,-37.676,-74.288,169.918,33.356,156.295
C06132=1046.877,-37.426,-74.301,169.920,33.357,156.295
C06133=1046.883,-37.177,-74.314,169.922,33.359,156.295
C06134=1046.889,-36.927,-74.327,169.924,33.360,156.295
C06135=1046.896,-36.678,-74.341,169.926,33.361,156.296
C06136=1046.902,-36.428,-74.354,169.928,33.362,156.296
C06137=1046.908,-36.178,-74.367,169.930,33.364,156.296
C06138=1046.914,-35.929,-74.380,169.932,33.365,156.296
C06139=1046.920,-35.680,-74.393,169.934,33.366,156.296
C06140=1046.927,-35.398,-74.408,169.936,33.368,156.296
C06141=1046.934,-35.118,-74.423,169.938,33.369,156.297
C06142=1046.942,-34.837,-74.438,169.940,33.370,156.297
C06143=1046.948,-34.556,-74.453,169.943,33.372,156.297
C06144=1046.954,-34.307,-74.466,169.945,33.373,156.297
C06145=1046.961,-34.057,-74.480,169.947,33.375,156.297
C06146=1046.967,-33.808,-74.493,169.949,33.376,156.298
C06147=1046.973,-33.558,-74.506,169.951,33.377,156.298
C06148=1046.979,-33.309,-74.519,169.953,33.378,156.298
C06149=1046.986,-33.059,-74.533,169.955,33.380,156.298
C06150=1046.992,-32.809,-74.546,169.957,33.381,156.298
C06151=1046.998,-32.560,-74.559,169.959,33.382,156.298
C06152=1047.005,-32.311,-74.572,169.961,33.383,156.298
C06153=1047.011,-32.061,-74.586,169.963,33.385,156.299
C06154=1047.018,-31.812,-74.599,169.965,33.386,156.299
C06155=1047.023,-31.562,-74.613,169.967,33.388,156.299
C06156=1047.030,-31.311,-74.626,169.969,33.388,156.299
C06157=1047.036,-31.062,-74.639,169.970,33.390,156.299
C06158=1047.042,-30.813,-74.653,169.972,33.391,156.299
C06159=1047.048,-30.564,-74.666,169.974,33.393,156.300
C06160=1047.055,-30.314,-74.680,169.976,33.394,156.300
C06161=1047.061,-30.064,-74.693,169.978,33.396,156.300
C06162=1047.067,-29.815,-74.706,169.980,33.396,156.300
C06163=1047.074,-29.565,-74.720,169.982,33.398,156.300
C06164=1047.080,-29.316,-74.734,169.984,33.399,156.300
C06165=1047.086,-29.066,-74.747,169.986,33.401,156.301
C06166=1047.093,-28.816,-74.760,169.988,33.402,156.301
C06167=1047.099,-28.567,-74.774,169.990,33.403,156.301
C06168=1047.106,-28.317,-74.787,169.992,33.404,156.301
C06169=1047.112,-28.068,-74.801,169.994,33.406,156.301
C06170=1047.118,-27.819,-74.814,169.996,33.407,156.302
C06171=1047.124,-27.568,-74.828,169.998,33.408,156.302
C06172=1047.131,-27.319,-74.841,170.000,33.410,156.302
C06173=1047.137,-27.070,-74.855,170.002,33.411,156.302
C06174=1047.144,-26.820,-74.868,170.004,33.412,156.302
C06175=1047.150,-26.571,-74.882,170.006,33.413,156.302
C06176=1047.155,-26.321,-74.895,170.008,33.415,156.303
C06177=1047.162,-26.071,-74.909,170.010,33.416,156.303
C06178=1047.168,-25.822,-74.922,170.012,33.418,156.303
C06179=1047.175,-25.572,-74.937,170.014,33.419,156.303
C06180=1047.181,-25.323,-74.951,170.016,33.421,156.303
C06181=1047.186,-25.073,-74.964,170.018,33.422,156.303
C06182=1047.193,-24.823,-74.978,170.020,33.423,156.304
C06183=1047.199,-24.574,-74.991,170.022,33.425,156.304
C06184=1047.205,-24.324,-75.005,170.023,33.426,156.304
C06185=1047.212,-24.075,-75.019,170.025,33.428,156.304
C06186=1047.218,-23.826,-75.033,170.027,33.429,156.304
C06187=1047.224,-23.576,-75.047,170.029,33.430,156.305
C06188=1047.230,-23.326,-75.060,170.031,33.432,156.305
C06189=1047.236,-23.077,-75.074,170.033,33.433,156.305
C06190=1047.243,-22.827,-75.088,170.035,33.435,156.305
C06191=1047.249,-22.578,-75.102,170.037,33.436,156.305
C06192=1047.255,-22.328,-75.116,170.039,33.438,156.306
C06193=1047.262,-22.079,-75.129,170.041,33.439,156.306
C06194=1047.268,-21.829,-75.143,170.043,33.440,156.306
C06195=1047.274,-21.580,-75.158,170.045,33.442,156.306
C06196=1047.280,-21.330,-75.171,170.047,33.443,156.306
C06197=1047.286,-21.080,-75.185,170.049,33.445,156.307
C06198=1047.293,-20.831,-75.198,170.050,33.446,156.307
C06199=1047.300,-20.582,-75.213,170.052,33.447,156.307
C06200=1047.305,-20.332,-75.227,170.054,33.449,156.307
C06201=1047.312,-20.082,-75.240,170.056,33.450,156.307
C06202=1047.318,-19.833,-75.255,170.058,33.452,156.307
C06203=1047.325,-19.583,-75.268,170.060,33.453,156.308
C06204=1047.332,-19.302,-75.284,170.062,33.455,156.308
C06205=1047.338,-19.020,-75.299,170.064,33.456,156.308
C06206=1047.346,-18.738,-75.315,170.067,33.458,156.308
C06207=1047.353,-18.457,-75.331,170.069,33.459,156.309
C06208=1047.359,-18.208,-75.344,170.071,33.461,156.309
C06209=1047.365,-17.958,-75.359,170.073,33.462,156.309
C06210=1047.372,-17.709,-75.372,170.074,33.464,156.309
C06211=1047.378,-17.459,-75.387,170.076,33.465,156.309
C06212=1047.384,-17.210,-75.401,170.078,33.466,156.310
C06213=1047.390,-16.960,-75.415,170.080,33.468,156.310
C06214=1047.397,-16.711,-75.429,170.082,33.469,156.310
C06215=1047.404,-16.461,-75.443,170.084,33.471,156.310
C06216=1047.410,-16.212,-75.457,170.086,33.473,156.310
C06217=1047.416,-15.962,-75.471,170.088,33.474,156.311
C06218=1047.422,-15.712,-75.485,170.090,33.475,156.311
C06219=1047.429,-15.463,-75.499,170.092,33.477,156.311
C06220=1047.435,-15.213,-75.513,170.094,33.478,156.311
C06221=1047.441,-14.965,-75.527,170.095,33.480,156.311
C06222=1047.447,-14.714,-75.541,170.097,33.481,156.312
C06223=1047.454,-14.465,-75.556,170.099,33.482,156.312
C06224=1047.460,-14.215,-75.570,170.101,33.484,156.312
C06225=1047.466,-13.966,-75.585,170.103,33.486,156.312
C06226=1047.472,-13.716,-75.598,170.105,33.487,156.312
C06227=1047.479,-13.467,-75.613,170.107,33.489,156.313
C06228=1047.484,-13.217,-75.627,170.109,33.490,156.313
C06229=1047.491,-12.968,-75.642,170.110,33.491,156.313
C06230=1047.497,-12.718,-75.655,170.112,33.493,156.313
C06231=1047.503,-12.469,-75.670,170.114,33.495,156.313
C06232=1047.509,-12.220,-75.684,170.116,33.496,156.314
C06233=1047.516,-11.970,-75.698,170.118,33.498,156.314
C06234=1047.522,-11.720,-75.713,170.120,33.499,156.314
C06235=1047.528,-11.470,-75.727,170.122,33.501,156.314
C06236=1047.535,-11.221,-75.741,170.124,33.502,156.314
C06237=1047.541,-10.972,-75.756,170.125,33.504,156.315
C06238=1047.547,-10.722,-75.770,170.127,33.505,156.315
C06239=1047.554,-10.473,-75.784,170.129,33.507,156.315
C06240=1047.559,-10.223,-75.798,170.131,33.508,156.315
C06241=1047.566,-9.973,-75.813,170.133,33.510,156.316
C06242=1047.572,-9.724,-75.828,170.135,33.512,156.316
C06243=1047.578,-9.474,-75.841,170.137,33.513,156.316
C06244=1047.585,-9.225,-75.856,170.138,33.514,156.316
C06245=1047.591,-8.976,-75.871,170.140,33.516,156.316
C06246=1047.597,-8.726,-75.885,170.142,33.517,156.317
C06247=1047.603,-8.477,-75.899,170.144,33.519,156.317
C06248=1047.610,-8.227,-75.914,170.146,33.521,156.317
C06249=1047.616,-7.978,-75.929,170.148,33.522,156.317
C06250=1047.622,-7.728,-75.942,170.150,33.523,156.318
C06251=1047.629,-7.479,-75.957,170.151,33.525,156.318
C06252=1047.635,-7.229,-75.972,170.153,33.527,156.318
C06253=1047.641,-6.980,-75.985,170.155,33.528,156.318
C06254=1047.648,-6.730,-76.000,170.157,33.530,156.318
C06255=1047.654,-6.480,-76.015,170.159,33.531,156.319
C06256=1047.660,-6.231,-76.030,170.161,33.532,156.319
C06257=1047.667,-5.981,-76.044,170.163,33.534,156.319
C06258=1047.673,-5.732,-76.059,170.164,33.536,156.319
C06259=1047.679,-5.482,-76.073,170.166,33.537,156.319
C06260=1047.685,-5.233,-76.088,170.168,33.539,156.320
C06261=1047.692,-4.984,-76.102,170.170,33.540,156.320
C06262=1047.698,-4.734,-76.117,170.172,33.542,156.320
C06263=1047.704,-4.485,-76.131,170.174,33.543,156.320
C06264=1047.711,-4.235,-76.146,170.176,33.545,156.321
C06265=1047.718,-3.986,-76.160,170.177,33.546,156.321
C06266=1047.724,-3.736,-76.175,170.179,33.548,156.321
C06267=1047.730,-3.487,-76.190,170.181,33.550,156.321
C06268=1047.737,-3.204,-76.206,170.183,33.551,156.321
C06269=1047.744,-2.921,-76.223,170.185,33.553,156.322
C06270=1047.751,-2.637,-76.240,170.187,33.555,156.322
C06271=1047.759,-2.354,-76.257,170.189,33.556,156.322
C06272=1047.764,-2.105,-76.272,170.191,33.558,156.323
C06273=1047.770,-1.855,-76.287,170.193,33.560,156.323
C06274=1047.776,-1.606,-76.302,170.195,33.561,156.323
C06275=1047.782,-1.356,-76.316,170.197,33.563,156.323
C06276=1047.788,-1.107,-76.331,170.198,33.565,156.323
C06277=1047.795,-0.857,-76.346,170.200,33.567,156.324
C06278=1047.800,-0.608,-76.360,170.202,33.568,156.324
C06279=1047.807,-0.358,-76.375,170.204,33.569,156.324
C06280=1047.813,-0.109,-76.390,170.206,33.571,156.324
C06281=1047.820,0.141,-76.405,170.207,33.573,156.325
C06282=1047.825,0.390,-76.420,170.209,33.575,156.325
C06283=1047.832,0.640,-76.435,170.211,33.576,156.325
C06284=1047.838,0.889,-76.450,170.213,33.578,156.325
C06285=1047.845,1.139,-76.465,170.215,33.580,156.326
C06286=1047.851,1.387,-76.480,170.216,33.581,156.326
C06287=1047.857,1.637,-76.495,170.218,33.583,156.326
C06288=1047.863,1.887,-76.510,170.220,33.584,156.326
C06289=1047.870,2.136,-76.525,170.222,33.586,156.327
C06290=1047.875,2.386,-76.540,170.224,33.588,156.327
C06291=1047.881,2.635,-76.555,170.225,33.589,156.327
C06292=1047.888,2.885,-76.570,170.227,33.591,156.327
C06293=1047.894,3.135,-76.585,170.229,33.593,156.328
C06294=1047.900,3.384,-76.600,170.231,33.594,156.328
C06295=1047.906,3.633,-76.614,170.233,33.596,156.328
C06296=1047.913,3.883,-76.629,170.234,33.597,156.328
C06297=1047.919,4.132,-76.644,170.236,33.599,156.329
C06298=1047.926,4.381,-76.660,170.238,33.601,156.329
C06299=1047.932,4.631,-76.675,170.240,33.602,156.329
C06300=1047.938,4.880,-76.689,170.241,33.604,156.329
C06301=1047.944,5.130,-76.704,170.243,33.605,156.330
C06302=1047.950,5.380,-76.720,170.245,33.607,156.330
C06303=1047.956,5.629,-76.735,170.247,33.609,156.330
C06304=1047.963,5.878,-76.750,170.249,33.610,156.330
C06305=1047.969,6.128,-76.765,170.250,33.612,156.331
C06306=1047.975,6.377,-76.780,170.252,33.614,156.331
C06307=1047.981,6.627,-76.795,170.254,33.615,156.331
C06308=1047.988,6.876,-76.810,170.256,33.617,156.331
C06309=1047.995,7.125,-76.825,170.258,33.618,156.331
C06310=1048.001,7.375,-76.840,170.259,33.620,156.332
C06311=1048.007,7.625,-76.855,170.261,33.622,156.332
C06312=1048.013,7.875,-76.871,170.263,33.623,156.332
C06313=1048.020,8.124,-76.887,170.265,33.625,156.332
C06314=1048.026,8.373,-76.901,170.266,33.627,156.333
C06315=1048.032,8.622,-76.916,170.268,33.629,156.333
C06316=1048.038,8.872,-76.931,170.270,33.630,156.333
C06317=1048.045,9.121,-76.947,170.272,33.631,156.333
C06318=1048.051,9.371,-76.962,170.274,33.633,156.334
C06319=1048.058,9.620,-76.977,170.275,33.635,156.334
C06320=1048.064,9.870,-76.993,170.278,33.637,156.334
C06321=1048.070,10.119,-77.008,170.280,33.638,156.334
C06322=1048.076,10.369,-77.023,170.282,33.640,156.335
C06323=1048.083,10.619,-77.038,170.283,33.641,156.335
C06324=1048.089,10.868,-77.053,170.285,33.643,156.335
C06325=1048.096,11.117,-77.068,170.287,33.645,156.335
C06326=1048.102,11.367,-77.083,170.289,33.646,156.336
C06327=1048.108,11.616,-77.099,170.291,33.648,156.336
C06328=1048.115,11.866,-77.114,170.292,33.650,156.336
C06329=1048.121,12.115,-77.130,170.294,33.651,156.336
C06330=1048.128,12.365,-77.145,170.296,33.653,156.337
C06331=1048.133,12.614,-77.160,170.298,33.654,156.337
C06332=1048.141,12.899,-77.177,170.300,33.656,156.337
C06333=1048.148,13.184,-77.195,170.302,33.658,156.337
C06334=1048.155,13.469,-77.212,170.304,33.660,156.338
C06335=1048.163,13.754,-77.230,170.306,33.662,156.338
C06336=1048.170,14.003,-77.246,170.307,33.663,156.338
C06337=1048.175,14.253,-77.261,170.309,33.665,156.338
C06338=1048.182,14.502,-77.277,170.311,33.667,156.339
C06339=1048.188,14.751,-77.292,170.313,33.669,156.339
C06340=1048.194,15.001,-77.307,170.314,33.670,156.339
C06341=1048.201,15.250,-77.323,170.316,33.672,156.339
C06342=1048.206,15.500,-77.339,170.318,33.673,156.340
C06343=1048.213,15.749,-77.354,170.320,33.675,156.340
C06344=1048.220,15.999,-77.370,170.321,33.677,156.340
C06345=1048.225,16.248,-77.385,170.323,33.679,156.340
C06346=1048.232,16.498,-77.401,170.325,33.680,156.341
C06347=1048.238,16.748,-77.417,170.327,33.682,156.341
C06348=1048.244,16.997,-77.432,170.328,33.684,156.341
C06349=1048.251,17.246,-77.447,170.330,33.685,156.342
C06350=1048.257,17.496,-77.463,170.332,33.687,156.342
C06351=1048.263,17.745,-77.478,170.334,33.689,156.342
C06352=1048.269,17.995,-77.495,170.335,33.691,156.342
C06353=1048.276,18.244,-77.510,170.337,33.692,156.343
C06354=1048.282,18.493,-77.525,170.339,33.694,156.343
C06355=1048.288,18.743,-77.542,170.341,33.696,156.343
C06356=1048.294,18.992,-77.556,170.342,33.698,156.343
C06357=1048.300,19.242,-77.573,170.344,33.699,156.344
C06358=1048.307,19.491,-77.588,170.346,33.701,156.344
C06359=1048.313,19.740,-77.603,170.347,33.702,156.344
C06360=1048.319,19.990,-77.620,170.349,33.704,156.344
C06361=1048.326,20.239,-77.635,170.351,33.706,156.345
C06362=1048.332,20.489,-77.651,170.353,33.708,156.345
C06363=1048.338,20.738,-77.667,170.354,33.710,156.345
C06364=1048.344,20.987,-77.683,170.356,33.711,156.345
C06365=1048.350,21.237,-77.698,170.358,33.713,156.346
C06366=1048.357,21.486,-77.714,170.360,33.714,156.346
C06367=1048.363,21.735,-77.730,170.361,33.716,156.346
C06368=1048.369,21.984,-77.746,170.363,33.718,156.347
C06369=1048.376,22.235,-77.762,170.365,33.720,156.347
C06370=1048.382,22.484,-77.777,170.366,33.722,156.347
C06371=1048.388,22.733,-77.794,170.368,33.723,156.347
C06372=1048.395,22.983,-77.809,170.370,33.725,156.348
C06373=1048.401,23.232,-77.825,170.372,33.727,156.348
C06374=1048.407,23.482,-77.841,170.374,33.728,156.348
C06375=1048.413,23.731,-77.857,170.376,33.730,156.348
C06376=1048.419,23.980,-77.873,170.378,33.732,156.349
C06377=1048.426,24.230,-77.888,170.379,33.734,156.349
C06378=1048.431,24.479,-77.904,170.381,33.736,156.349
C06379=1048.438,24.728,-77.920,170.383,33.737,156.349
C06380=1048.445,24.978,-77.937,170.385,33.739,156.350
C06381=1048.451,25.228,-77.953,170.386,33.740,156.350
C06382=1048.457,25.477,-77.968,170.388,33.742,156.350
C06383=1048.463,25.727,-77.984,170.390,33.744,156.351
C06384=1048.470,25.976,-78.000,170.391,33.746,156.351
C06385=1048.476,26.225,-78.016,170.393,33.748,156.351
C06386=1048.482,26.474,-78.032,170.395,33.749,156.351
C06387=1048.489,26.724,-78.048,170.396,33.751,156.352
C06388=1048.495,26.973,-78.064,170.398,33.752,156.352
C06389=1048.502,27.223,-78.080,170.400,33.755,156.352
C06390=1048.507,27.472,-78.096,170.402,33.757,156.352
C06391=1048.513,27.722,-78.112,170.403,33.758,156.353
C06392=1048.520,27.971,-78.128,170.405,33.760,156.353
C06393=1048.526,28.221,-78.144,170.407,33.762,156.353
C06394=1048.532,28.470,-78.160,170.408,33.763,156.354
C06395=1048.539,28.719,-78.176,170.410,33.765,156.354
C06396=1048.546,29.006,-78.195,170.412,33.767,156.354
C06397=1048.552,29.291,-78.214,170.414,33.769,156.354
C06398=1048.560,29.578,-78.232,170.416,33.771,156.355
C06399=1048.567,29.865,-78.250,170.418,33.773,156.355
C06400=1048.573,30.113,-78.267,170.420,33.775,156.355
C06401=1048.579,30.363,-78.283,170.421,33.777,156.356
C06402=1048.586,30.612,-78.299,170.423,33.779,156.356
C06403=1048.592,30.862,-78.316,170.425,33.781,156.356
C06404=1048.598,31.111,-78.332,170.426,33.782,156.357
C06405=1048.604,31.360,-78.348,170.428,33.784,156.357
C06406=1048.610,31.610,-78.364,170.430,33.786,156.357
C06407=1048.618,31.859,-78.380,170.431,33.788,156.357
C06408=1048.623,32.109,-78.397,170.433,33.789,156.358
C06409=1048.629,32.358,-78.413,170.435,33.791,156.358
C06410=1048.635,32.608,-78.429,170.436,33.793,156.358
C06411=1048.641,32.857,-78.446,170.438,33.794,156.358
C06412=1048.648,33.107,-78.462,170.441,33.796,156.359
C06413=1048.655,33.356,-78.478,170.442,33.798,156.359
C06414=1048.661,33.605,-78.494,170.444,33.800,156.359
C06415=1048.666,33.855,-78.510,170.446,33.802,156.360
C06416=1048.673,34.104,-78.528,170.447,33.804,156.360
C06417=1048.679,34.353,-78.544,170.449,33.806,156.360
C06418=1048.685,34.603,-78.560,170.451,33.807,156.360
C06419=1048.692,34.852,-78.576,170.453,33.809,156.361
C06420=1048.698,35.102,-78.592,170.454,33.811,156.361
C06421=1048.704,35.351,-78.609,170.456,33.812,156.361
C06422=1048.711,35.600,-78.626,170.458,33.814,156.362
C06423=1048.717,35.849,-78.642,170.459,33.816,156.362
C06424=1048.723,36.099,-78.659,170.461,33.818,156.362
C06425=1048.730,36.348,-78.674,170.463,33.820,156.362
C06426=1048.736,36.598,-78.690,170.464,33.822,156.363
C06427=1048.742,36.847,-78.707,170.466,33.823,156.363
C06428=1048.749,37.096,-78.724,170.468,33.825,156.363
C06429=1048.755,37.346,-78.740,170.469,33.827,156.364
C06430=1048.761,37.595,-78.757,170.471,33.828,156.364
C06431=1048.767,37.845,-78.773,170.473,33.830,156.364
C06432=1048.773,38.094,-78.790,170.474,33.832,156.364
C06433=1048.779,38.343,-78.806,170.476,33.834,156.365
C06434=1048.785,38.593,-78.823,170.478,33.836,156.365
C06435=1048.792,38.842,-78.840,170.479,33.838,156.365
C06436=1048.798,39.091,-78.856,170.481,33.840,156.366
C06437=1048.804,39.341,-78.873,170.483,33.842,156.366
C06438=1048.811,39.591,-78.889,170.484,33.843,156.366
C06439=1048.817,39.840,-78.906,170.486,33.845,156.366
C06440=1048.823,40.089,-78.922,170.488,33.847,156.367
C06441=1048.829,40.338,-78.939,170.489,33.849,156.367
C06442=1048.836,40.588,-78.956,170.491,33.851,156.367
C06443=1048.842,40.837,-78.972,170.494,33.852,156.368
C06444=1048.848,41.086,-78.989,170.495,33.854,156.368
C06445=1048.854,41.336,-79.006,170.497,33.856,156.368
C06446=1048.860,41.585,-79.022,170.499,33.858,156.369
C06447=1048.866,41.834,-79.040,170.500,33.859,156.369
C06448=1048.872,42.084,-79.056,170.502,33.861,156.369
C06449=1048.878,42.334,-79.073,170.504,33.863,156.369
C06450=1048.885,42.582,-79.090,170.505,33.865,156.370
C06451=1048.891,42.832,-79.106,170.507,33.867,156.370
C06452=1048.897,43.081,-79.123,170.508,33.869,156.370
C06453=1048.904,43.331,-79.140,170.510,33.871,156.371
C06454=1048.910,43.580,-79.157,170.512,33.873,156.371
C06455=1048.916,43.829,-79.173,170.513,33.875,156.371
C06456=1048.922,44.078,-79.191,170.515,33.877,156.372
C06457=1048.928,44.328,-79.207,170.517,33.879,156.372
C06458=1048.934,44.577,-79.224,170.518,33.880,156.372
C06459=1048.940,44.827,-79.241,170.520,33.882,156.372
C06460=1048.947,45.112,-79.260,170.522,33.884,156.373
C06461=1048.955,45.400,-79.280,170.524,33.886,156.373
C06462=1048.962,45.686,-79.300,170.526,33.888,156.373
C06463=1048.968,45.972,-79.319,170.527,33.891,156.374
C06464=1048.975,46.221,-79.336,170.529,33.892,156.374
C06465=1048.980,46.470,-79.352,170.531,33.894,156.374
C06466=1048.987,46.720,-79.370,170.532,33.896,156.375
C06467=1048.993,46.969,-79.387,170.534,33.898,156.375
C06468=1048.999,47.218,-79.403,170.537,33.900,156.375
C06469=1049.005,47.468,-79.421,170.538,33.902,156.376
C06470=1049.011,47.717,-79.438,170.540,33.904,156.376
C06471=1049.018,47.967,-79.455,170.542,33.906,156.376
C06472=1049.023,48.216,-79.472,170.543,33.907,156.376
C06473=1049.029,48.465,-79.489,170.545,33.909,156.377
C06474=1049.036,48.714,-79.506,170.546,33.911,156.377
C06475=1049.041,48.964,-79.523,170.548,33.913,156.377
C06476=1049.048,49.213,-79.540,170.550,33.915,156.378
C06477=1049.054,49.463,-79.557,170.551,33.917,156.378
C06478=1049.060,49.712,-79.574,170.553,33.919,156.378
C06479=1049.066,49.961,-79.592,170.555,33.921,156.379
C06480=1049.072,50.211,-79.608,170.556,33.923,156.379
C06481=1049.079,50.460,-79.626,170.558,33.925,156.379
C06482=1049.085,50.709,-79.643,170.560,33.927,156.380
C06483=1049.092,50.958,-79.660,170.561,33.928,156.380
C06484=1049.097,51.208,-79.677,170.563,33.930,156.380
C06485=1049.103,51.457,-79.694,170.564,33.932,156.381
C06486=1049.110,51.706,-79.711,170.566,33.934,156.381
C06487=1049.115,51.956,-79.728,170.568,33.936,156.381
C06488=1049.122,52.205,-79.745,170.569,33.938,156.381
C06489=1049.128,52.454,-79.763,170.571,33.940,156.382
C06490=1049.134,52.704,-79.780,170.573,33.942,156.382
C06491=1049.140,52.953,-79.797,170.574,33.944,156.382
C06492=1049.147,53.203,-79.814,170.577,33.946,156.383
C06493=1049.153,53.452,-79.831,170.579,33.948,156.383
C06494=1049.160,53.701,-79.849,170.580,33.949,156.383
C06495=1049.165,53.950,-79.866,170.582,33.951,156.384
C06496=1049.172,54.200,-79.883,170.583,33.953,156.384
C06497=1049.177,54.449,-79.901,170.585,33.955,156.384
C06498=1049.184,54.699,-79.918,170.587,33.957,156.384
C06499=1049.190,54.947,-79.935,170.588,33.959,156.385
C06500=1049.196,55.197,-79.953,170.590,33.960,156.385
C06501=1049.202,55.446,-79.969,170.592,33.962,156.385
C06502=1049.209,55.696,-79.987,170.593,33.964,156.386
C06503=1049.215,55.945,-80.004,170.595,33.966,156.386
C06504=1049.222,56.194,-80.021,170.597,33.968,156.386
C06505=1049.227,56.443,-80.039,170.598,33.970,156.387
C06506=1049.234,56.693,-80.056,170.600,33.971,156.387
C06507=1049.241,56.942,-80.074,170.601,33.973,156.387
C06508=1049.246,57.192,-80.090,170.603,33.975,156.387
C06509=1049.253,57.441,-80.108,170.605,33.977,156.388
C06510=1049.258,57.690,-80.125,170.606,33.979,156.388
C06511=1049.265,57.940,-80.143,170.608,33.981,156.388
C06512=1049.271,58.189,-80.160,170.610,33.982,156.389
C06513=1049.278,58.438,-80.178,170.611,33.984,156.389
C06514=1049.285,58.688,-80.195,170.613,33.986,156.389
C06515=1049.290,58.937,-80.212,170.616,33.988,156.390
C06516=1049.297,59.186,-80.230,170.617,33.990,156.390
C06517=1049.302,59.435,-80.247,170.619,33.991,156.390
C06518=1049.309,59.685,-80.265,170.620,33.993,156.390
C06519=1049.316,59.934,-80.282,170.622,33.995,156.391
C06520=1049.322,60.183,-80.300,170.624,33.997,156.391
C06521=1049.329,60.433,-80.317,170.625,33.999,156.391
C06522=1049.334,60.682,-80.334,170.627,34.001,156.392
C06523=1049.341,60.931,-80.352,170.629,34.003,156.392
C06524=1049.348,61.217,-80.372,170.631,34.005,156.392
C06525=1049.355,61.503,-80.392,170.632,34.007,156.393
C06526=1049.362,61.790,-80.412,170.634,34.009,156.393
C06527=1049.370,62.075,-80.431,170.636,34.011,156.393
C06528=1049.376,62.325,-80.449,170.638,34.013,156.394
C06529=1049.382,62.574,-80.466,170.640,34.015,156.394
C06530=1049.389,62.823,-80.485,170.641,34.016,156.394
C06531=1049.396,63.072,-80.502,170.643,34.018,156.395
C06532=1049.401,63.321,-80.520,170.644,34.020,156.395
C06533=1049.408,63.571,-80.537,170.646,34.022,156.395
C06534=1049.414,63.820,-80.555,170.648,34.024,156.396
C06535=1049.421,64.069,-80.572,170.649,34.026,156.396
C06536=1049.427,64.319,-80.590,170.652,34.028,156.396
C06537=1049.434,64.568,-80.607,170.654,34.030,156.396
C06538=1049.439,64.817,-80.625,170.655,34.031,156.397
C06539=1049.445,65.067,-80.643,170.657,34.033,156.397
C06540=1049.452,65.316,-80.662,170.659,34.035,156.397
C06541=1049.458,65.565,-80.679,170.660,34.037,156.398
C06542=1049.464,65.815,-80.696,170.662,34.039,156.398
C06543=1049.470,66.064,-80.714,170.663,34.041,156.398
C06544=1049.476,66.313,-80.731,170.665,34.043,156.399
C06545=1049.483,66.562,-80.750,170.667,34.045,156.399
C06546=1049.489,66.812,-80.768,170.668,34.047,156.399
C06547=1049.495,67.061,-80.785,170.670,34.048,156.399
C06548=1049.501,67.310,-80.803,170.672,34.050,156.400
C06549=1049.507,67.560,-80.821,170.673,34.052,156.400
C06550=1049.513,67.809,-80.839,170.675,34.054,156.400
C06551=1049.520,68.058,-80.856,170.676,34.056,156.401
C06552=1049.527,68.328,-80.876,170.678,34.058,156.401
C06553=1049.533,68.596,-80.895,170.680,34.060,156.401
C06554=1049.540,68.866,-80.915,170.682,34.063,156.402
C06555=1049.547,69.134,-80.933,170.684,34.065,156.402
C06556=1049.553,69.384,-80.951,170.686,34.067,156.403
C06557=1049.559,69.633,-80.970,170.688,34.069,156.403
C06558=1049.565,69.883,-80.988,170.689,34.071,156.403
C06559=1049.571,70.132,-81.005,170.691,34.073,156.403
C06560=1049.577,70.381,-81.024,170.692,34.074,156.404
C06561=1049.584,70.630,-81.041,170.694,34.076,156.404
C06562=1049.590,70.879,-81.059,170.696,34.078,156.404
C06563=1049.596,71.129,-81.078,170.697,34.080,156.405
C06564=1049.602,71.378,-81.096,170.699,34.082,156.405
C06565=1049.608,71.628,-81.114,170.701,34.084,156.405
C06566=1049.614,71.876,-81.132,170.702,34.086,156.406
C06567=1049.620,72.126,-81.150,170.704,34.087,156.406
C06568=1049.627,72.375,-81.168,170.705,34.089,156.406
C06569=1049.632,72.624,-81.186,170.707,34.091,156.407
C06570=1049.638,72.873,-81.205,170.709,34.093,156.407
C06571=1049.645,73.123,-81.222,170.710,34.095,156.407
C06572=1049.651,73.373,-81.240,170.712,34.097,156.408
C06573=1049.657,73.621,-81.258,170.714,34.099,156.408
C06574=1049.663,73.871,-81.276,170.716,34.101,156.408
C06575=1049.670,74.120,-81.295,170.718,34.103,156.409
C06576=1049.676,74.370,-81.313,170.719,34.105,156.409
C06577=1049.682,74.618,-81.331,170.721,34.107,156.409
C06578=1049.688,74.868,-81.349,170.723,34.109,156.410
C06579=1049.694,75.117,-81.368,170.724,34.111,156.410
C06580=1049.700,75.367,-81.385,170.726,34.113,156.410
C06581=1049.707,75.616,-81.404,170.727,34.115,156.411
C06582=1049.712,75.865,-81.422,170.729,34.117,156.411
C06583=1049.719,76.114,-81.440,170.731,34.119,156.411
C06584=1049.725,76.364,-81.458,170.732,34.121,156.412
C06585=1049.731,76.613,-81.477,170.734,34.123,156.412
C06586=1049.738,76.862,-81.494,170.736,34.125,156.412
C06587=1049.744,77.111,-81.513,170.737,34.126,156.412
C06588=1049.751,77.377,-81.532,170.739,34.128,156.413
C06589=1049.757,77.643,-81.552,170.741,34.130,156.413
C06590=1049.764,77.910,-81.572,170.743,34.132,156.413
C06591=1049.771,78.174,-81.591,170.745,34.134,156.414
C06592=1049.777,78.424,-81.609,170.747,34.136,156.414
C06593=1049.783,78.673,-81.627,170.748,34.138,156.414
C06594=1049.788,78.923,-81.646,170.750,34.141,156.415
C06595=1049.794,79.172,-81.665,170.752,34.143,156.415
C06596=1049.801,79.421,-81.683,170.753,34.145,156.416
C06597=1049.807,79.671,-81.701,170.755,34.147,156.416
C06598=1049.813,79.920,-81.720,170.756,34.148,156.416
C06599=1049.819,80.169,-81.739,170.758,34.150,156.417
C06600=1049.825,80.418,-81.757,170.760,34.152,156.417
C06601=1049.831,80.667,-81.775,170.761,34.154,156.417
C06602=1049.837,80.917,-81.794,170.763,34.156,156.417
C06603=1049.844,81.166,-81.813,170.764,34.158,156.418
C06604=1049.849,81.415,-81.830,170.766,34.160,156.418
C06605=1049.855,81.664,-81.849,170.768,34.162,156.418
C06606=1049.862,81.913,-81.868,170.770,34.164,156.419
C06607=1049.868,82.162,-81.887,170.772,34.166,156.419
C06608=1049.874,82.412,-81.905,170.774,34.168,156.419
C06609=1049.881,82.661,-81.923,170.775,34.170,156.420
C06610=1049.886,82.911,-81.943,170.777,34.172,156.420
C06611=1049.892,83.159,-81.961,170.778,34.174,156.420
C06612=1049.898,83.409,-81.979,170.780,34.176,156.421
C06613=1049.905,83.658,-81.997,170.782,34.178,156.421
C06614=1049.910,83.907,-82.017,170.783,34.180,156.422
C06615=1049.917,84.156,-82.035,170.785,34.182,156.422
C06616=1049.923,84.406,-82.054,170.787,34.184,156.422
C06617=1049.929,84.655,-82.072,170.788,34.186,156.423
C06618=1049.936,84.904,-82.091,170.790,34.188,156.423
C06619=1049.941,85.154,-82.110,170.791,34.190,156.423
C06620=1049.947,85.402,-82.128,170.793,34.192,156.423
C06621=1049.954,85.651,-82.147,170.795,34.194,156.424
C06622=1049.960,85.901,-82.165,170.797,34.196,156.424
C06623=1049.966,86.150,-82.185,170.799,34.198,156.424
C06624=1049.972,86.400,-82.203,170.801,34.200,156.425
C06625=1049.978,86.649,-82.221,170.802,34.202,156.425
C06626=1049.985,86.898,-82.240,170.804,34.204,156.425
C06627=1049.990,87.147,-82.259,170.805,34.205,156.426
C06628=1049.997,87.397,-82.278,170.807,34.207,156.426
C06629=1050.003,87.646,-82.296,170.809,34.209,156.426
C06630=1050.010,87.895,-82.315,170.810,34.211,156.427
C06631=1050.015,88.144,-82.334,170.812,34.213,156.427
C06632=1050.022,88.393,-82.353,170.814,34.215,156.427
C06633=1050.028,88.642,-82.372,170.815,34.217,156.428
C06634=1050.035,88.892,-82.390,170.817,34.219,156.428
C06635=1050.040,89.141,-82.409,170.818,34.221,156.428
C06636=1050.047,89.390,-82.428,170.820,34.223,156.429
C06637=1050.053,89.640,-82.446,170.823,34.225,156.429
C06638=1050.059,89.889,-82.465,170.824,34.227,156.429
C06639=1050.065,90.138,-82.484,170.826,34.229,156.430
C06640=1050.071,90.388,-82.503,170.828,34.231,156.430
C06641=1050.078,90.637,-82.521,170.829,34.233,156.430
C06642=1050.084,90.885,-82.541,170.831,34.235,156.431
C06643=1050.090,91.135,-82.560,170.833,34.237,156.431
C06644=1050.096,91.384,-82.579,170.834,34.238,156.431
C06645=1050.102,91.633,-82.598,170.836,34.240,156.432
C06646=1050.108,91.883,-82.617,170.837,34.243,156.432
C06647=1050.114,92.132,-82.636,170.839,34.245,156.432
C06648=1050.120,92.381,-82.655,170.841,34.247,156.433
C06649=1050.127,92.630,-82.674,170.842,34.249,156.433
C06650=1050.132,92.879,-82.692,170.844,34.251,156.433
C06651=1050.138,93.128,-82.711,170.846,34.253,156.434
C06652=1050.146,93.414,-82.733,170.848,34.255,156.434
C06653=1050.153,93.700,-82.755,170.850,34.257,156.435
C06654=1050.159,93.985,-82.778,170.852,34.260,156.435
C06655=1050.166,94.272,-82.799,170.854,34.262,156.435
C06656=1050.173,94.520,-82.819,170.856,34.264,156.436
C06657=1050.178,94.770,-82.838,170.857,34.266,156.436
C06658=1050.185,95.019,-82.856,170.859,34.268,156.436
C06659=1050.190,95.268,-82.876,170.861,34.270,156.437
C06660=1050.197,95.517,-82.894,170.862,34.272,156.437
C06661=1050.203,95.766,-82.914,170.864,34.274,156.437
C06662=1050.209,96.015,-82.933,170.865,34.276,156.438
C06663=1050.215,96.265,-82.952,170.867,34.278,156.438
C06664=1050.221,96.514,-82.971,170.869,34.280,156.438
C06665=1050.227,96.763,-82.990,170.871,34.282,156.439
C06666=1050.234,97.012,-83.009,170.873,34.284,156.439
C06667=1050.240,97.261,-83.029,170.875,34.285,156.439
C06668=1050.245,97.511,-83.048,170.876,34.287,156.440
C06669=1050.252,97.760,-83.067,170.878,34.290,156.440
C06670=1050.258,98.009,-83.087,170.880,34.292,156.440
C06671=1050.264,98.258,-83.105,170.881,34.294,156.441
C06672=1050.270,98.508,-83.125,170.883,34.296,156.441
C06673=1050.277,98.756,-83.144,170.884,34.298,156.441
C06674=1050.283,99.006,-83.163,170.886,34.300,156.442
C06675=1050.289,99.255,-83.182,170.888,34.302,156.442
C06676=1050.295,99.504,-83.202,170.889,34.303,156.442
C06677=1050.301,99.753,-83.221,170.891,34.305,156.443
C06678=1050.307,100.002,-83.240,170.893,34.307,156.443
C06679=1050.313,100.251,-83.260,170.895,34.309,156.443
C06680=1050.320,100.500,-83.279,170.897,34.311,156.444
C06681=1050.326,100.750,-83.298,170.899,34.313,156.444
C06682=1050.332,100.999,-83.318,170.900,34.316,156.445
C06683=1050.338,101.249,-83.337,170.902,34.318,156.445
C06684=1050.344,101.497,-83.357,170.904,34.320,156.445
C06685=1050.350,101.747,-83.376,170.905,34.321,156.446
C06686=1050.356,101.996,-83.395,170.907,34.323,156.446
C06687=1050.362,102.245,-83.415,170.909,34.325,156.446
C06688=1050.367,102.494,-83.434,170.910,34.328,156.447
C06689=1050.374,102.743,-83.454,170.912,34.330,156.447
C06690=1050.380,102.993,-83.473,170.913,34.332,156.447
C06691=1050.386,103.242,-83.493,170.915,34.334,156.448
C06692=1050.392,103.491,-83.513,170.918,34.336,156.448
C06693=1050.398,103.740,-83.533,170.919,34.338,156.448
C06694=1050.405,103.989,-83.551,170.921,34.340,156.449
C06695=1050.411,104.238,-83.571,170.923,34.342,156.449
C06696=1050.416,104.487,-83.590,170.924,34.344,156.449
C06697=1050.422,104.736,-83.610,170.926,34.346,156.450
C06698=1050.429,104.986,-83.630,170.928,34.348,156.450
C06699=1050.435,105.235,-83.650,170.929,34.350,156.450
C06700=1050.441,105.484,-83.669,170.931,34.352,156.451
C06701=1050.447,105.733,-83.689,170.933,34.354,156.451
C06702=1050.453,105.982,-83.708,170.934,34.356,156.452
C06703=1050.459,106.231,-83.728,170.936,34.358,156.452
C06704=1050.465,106.481,-83.748,170.939,34.360,156.452
C06705=1050.471,106.730,-83.767,170.940,34.362,156.453
C06706=1050.478,106.979,-83.787,170.942,34.364,156.453
C06707=1050.483,107.228,-83.806,170.944,34.366,156.453
C06708=1050.489,107.477,-83.826,170.945,34.368,156.454
C06709=1050.496,107.726,-83.846,170.947,34.370,156.454
C06710=1050.502,107.976,-83.865,170.949,34.372,156.454
C06711=1050.508,108.225,-83.885,170.950,34.374,156.455
C06712=1050.514,108.473,-83.905,170.952,34.376,156.455
C06713=1050.521,108.723,-83.924,170.954,34.378,156.455
C06714=1050.527,108.972,-83.944,170.955,34.381,156.456
C06715=1050.532,109.222,-83.964,170.957,34.382,156.456
C06716=1050.540,109.507,-83.987,170.959,34.384,156.456
C06717=1050.547,109.793,-84.010,170.962,34.387,156.457
C06718=1050.554,110.078,-84.032,170.964,34.389,156.457
C06719=1050.560,110.364,-84.054,170.966,34.391,156.458
C06720=1050.567,110.613,-84.075,170.967,34.393,156.458
C06721=1050.573,110.863,-84.094,170.969,34.395,156.458
C06722=1050.579,111.111,-84.114,170.971,34.397,156.459
C06723=1050.585,111.360,-84.134,170.972,34.400,156.459
C06724=1050.591,111.610,-84.154,170.974,34.402,156.459
C06725=1050.597,111.859,-84.174,170.976,34.404,156.460
C06726=1050.603,112.108,-84.194,170.977,34.406,156.460
C06727=1050.609,112.357,-84.213,170.979,34.407,156.460
C06728=1050.615,112.606,-84.234,170.982,34.410,156.461
C06729=1050.621,112.855,-84.254,170.983,34.412,156.461
C06730=1050.627,113.105,-84.273,170.985,34.414,156.461
C06731=1050.634,113.354,-84.293,170.987,34.416,156.462
C06732=1050.640,113.603,-84.313,170.988,34.418,156.462
C06733=1050.646,113.852,-84.333,170.990,34.420,156.463
C06734=1050.652,114.101,-84.353,170.992,34.422,156.463
C06735=1050.658,114.350,-84.374,170.993,34.424,156.463
C06736=1050.664,114.599,-84.394,170.995,34.426,156.464
C06737=1050.669,114.849,-84.413,170.997,34.429,156.464
C06738=1050.675,115.097,-84.433,170.998,34.430,156.464
C06739=1050.682,115.347,-84.454,171.000,34.432,156.465
C06740=1050.687,115.596,-84.474,171.003,34.435,156.465
C06741=1050.693,115.845,-84.494,171.004,34.437,156.466
C06742=1050.699,116.094,-84.514,171.006,34.439,156.466
C06743=1050.706,116.343,-84.534,171.008,34.441,156.466
C06744=1050.711,116.592,-84.555,171.009,34.443,156.467
C06745=1050.717,116.841,-84.575,171.011,34.445,156.467
C06746=1050.724,117.091,-84.595,171.013,34.447,156.467
C06747=1050.730,117.339,-84.615,171.014,34.450,156.468
C06748=1050.735,117.589,-84.636,171.016,34.452,156.468
C06749=1050.741,117.837,-84.656,171.018,34.453,156.468
C06750=1050.747,118.087,-84.676,171.020,34.456,156.469
C06751=1050.753,118.336,-84.697,171.022,34.458,156.469
C06752=1050.759,118.585,-84.717,171.024,34.460,156.470
C06753=1050.765,118.834,-84.737,171.025,34.462,156.470
C06754=1050.771,119.083,-84.757,171.027,34.464,156.470
C06755=1050.776,119.332,-84.777,171.029,34.466,156.471
C06756=1050.783,119.582,-84.798,171.031,34.468,156.471
C06757=1050.789,119.831,-84.818,171.032,34.471,156.471
C06758=1050.794,120.080,-84.838,171.034,34.473,156.472
C06759=1050.801,120.329,-84.859,171.036,34.475,156.472
C06760=1050.807,120.577,-84.879,171.037,34.476,156.472
C06761=1050.813,120.826,-84.899,171.040,34.479,156.473
C06762=1050.819,121.076,-84.920,171.042,34.481,156.473
C06763=1050.825,121.325,-84.940,171.043,34.483,156.474
C06764=1050.832,121.574,-84.960,171.045,34.485,156.474
C06765=1050.837,121.824,-84.981,171.047,34.487,156.474
C06766=1050.843,122.072,-85.001,171.049,34.489,156.475
C06767=1050.849,122.322,-85.021,171.050,34.491,156.475
C06768=1050.855,122.570,-85.042,171.052,34.493,156.475
C06769=1050.862,122.820,-85.063,171.054,34.496,156.476
C06770=1050.868,123.069,-85.083,171.055,34.497,156.476
C06771=1050.873,123.318,-85.103,171.057,34.499,156.476
C06772=1050.879,123.567,-85.124,171.060,34.501,156.477
C06773=1050.886,123.816,-85.144,171.062,34.504,156.477
C06774=1050.892,124.065,-85.165,171.063,34.506,156.478
C06775=1050.898,124.314,-85.185,171.065,34.508,156.478
C06776=1050.904,124.563,-85.205,171.067,34.510,156.478
C06777=1050.909,124.813,-85.226,171.068,34.512,156.479
C06778=1050.916,125.061,-85.247,171.070,34.514,156.479
C06779=1050.922,125.311,-85.267,171.072,34.516,156.479
C06780=1050.929,125.596,-85.291,171.074,34.519,156.480
C06781=1050.936,125.882,-85.314,171.076,34.521,156.480
C06782=1050.943,126.167,-85.337,171.078,34.523,156.481
C06783=1050.950,126.453,-85.361,171.081,34.526,156.481
C06784=1050.957,126.702,-85.381,171.082,34.527,156.481
C06785=1050.962,126.951,-85.403,171.084,34.530,156.482
C06786=1050.969,127.200,-85.423,171.086,34.532,156.482
C06787=1050.974,127.449,-85.443,171.088,34.534,156.482
C06788=1050.981,127.698,-85.464,171.089,34.536,156.483
C06789=1050.987,127.947,-85.484,171.091,34.538,156.483
C06790=1050.993,128.197,-85.505,171.093,34.540,156.484
C06791=1050.999,128.445,-85.526,171.095,34.542,156.484
C06792=1051.006,128.695,-85.546,171.096,34.544,156.484
C06793=1051.011,128.944,-85.567,171.099,34.546,156.485
C06794=1051.018,129.193,-85.588,171.101,34.548,156.485
C06795=1051.024,129.441,-85.608,171.103,34.550,156.485
C06796=1051.030,129.691,-85.630,171.104,34.552,156.486
C06797=1051.036,129.939,-85.650,171.106,34.554,156.486
C06798=1051.042,130.189,-85.670,171.108,34.556,156.486
C06799=1051.048,130.437,-85.691,171.110,34.559,156.487
C06800=1051.055,130.687,-85.711,171.111,34.561,156.487
C06801=1051.061,130.936,-85.733,171.113,34.563,156.487
C06802=1051.067,131.185,-85.753,171.115,34.564,156.488
C06803=1051.074,131.434,-85.774,171.118,34.566,156.488
C06804=1051.079,131.683,-85.795,171.119,34.569,156.489
C06805=1051.085,131.932,-85.816,171.121,34.571,156.489
C06806=1051.091,132.181,-85.836,171.123,34.573,156.489
C06807=1051.097,132.430,-85.858,171.125,34.575,156.490
C06808=1051.103,132.679,-85.878,171.126,34.577,156.490
C06809=1051.110,132.928,-85.899,171.128,34.580,156.491
C06810=1051.115,133.177,-85.920,171.130,34.582,156.491
C06811=1051.121,133.427,-85.942,171.132,34.584,156.491
C06812=1051.128,133.676,-85.962,171.133,34.586,156.492
C06813=1051.133,133.925,-85.983,171.136,34.588,156.492
C06814=1051.139,134.174,-86.005,171.138,34.590,156.492
C06815=1051.145,134.423,-86.025,171.140,34.592,156.493
C06816=1051.151,134.672,-86.046,171.142,34.594,156.493
C06817=1051.157,134.921,-86.067,171.143,34.596,156.493
C06818=1051.164,135.170,-86.088,171.145,34.599,156.494
C06819=1051.170,135.419,-86.110,171.147,34.601,156.494
C06820=1051.175,135.668,-86.130,171.149,34.603,156.495
C06821=1051.182,135.917,-86.151,171.150,34.605,156.495
C06822=1051.188,136.166,-86.173,171.152,34.607,156.495
C06823=1051.193,136.415,-86.193,171.155,34.609,156.496
C06824=1051.200,136.665,-86.215,171.157,34.611,156.496
C06825=1051.206,136.913,-86.236,171.158,34.613,156.496
C06826=1051.212,137.163,-86.257,171.160,34.616,156.497
C06827=1051.217,137.411,-86.278,171.162,34.618,156.497
C06828=1051.224,137.660,-86.299,171.164,34.620,156.498
C06829=1051.230,137.910,-86.320,171.166,34.622,156.498
C06830=1051.236,138.158,-86.341,171.167,34.624,156.498
C06831=1051.242,138.408,-86.363,171.169,34.626,156.499
C06832=1051.248,138.656,-86.384,171.172,34.629,156.499
C06833=1051.254,138.906,-86.404,171.174,34.631,156.500
C06834=1051.260,139.155,-86.426,171.175,34.632,156.500
C06835=1051.266,139.403,-86.447,171.177,34.635,156.500
C06836=1051.273,139.652,-86.468,171.179,34.637,156.501
C06837=1051.279,139.901,-86.490,171.181,34.639,156.501
C06838=1051.284,140.151,-86.511,171.183,34.641,156.501
C06839=1051.290,140.400,-86.532,171.184,34.643,156.502
C06840=1051.296,140.649,-86.554,171.186,34.646,156.502
C06841=1051.302,140.897,-86.575,171.188,34.648,156.503
C06842=1051.308,141.147,-86.597,171.191,34.650,156.503
C06843=1051.314,141.396,-86.618,171.193,34.652,156.503
C06844=1051.321,141.681,-86.642,171.195,34.655,156.504
C06845=1051.328,141.966,-86.667,171.197,34.657,156.504
C06846=1051.334,142.252,-86.691,171.199,34.660,156.505
C06847=1051.341,142.537,-86.716,171.201,34.662,156.505
C06848=1051.347,142.786,-86.737,171.203,34.664,156.506
C06849=1051.354,143.035,-86.759,171.204,34.667,156.506
C06850=1051.359,143.284,-86.780,171.207,34.669,156.506
C06851=1051.365,143.533,-86.802,171.209,34.671,156.507
C06852=1051.372,143.782,-86.823,171.211,34.673,156.507
C06853=1051.377,144.031,-86.845,171.213,34.675,156.507
C06854=1051.383,144.280,-86.866,171.214,34.677,156.508
C06855=1051.389,144.529,-86.888,171.216,34.679,156.508
C06856=1051.396,144.778,-86.910,171.218,34.682,156.509
C06857=1051.401,145.027,-86.931,171.220,34.684,156.509
C06858=1051.407,145.276,-86.953,171.222,34.686,156.509
C06859=1051.413,145.525,-86.974,171.224,34.688,156.510
C06860=1051.420,145.774,-86.995,171.226,34.690,156.510
C06861=1051.426,146.023,-87.016,171.228,34.693,156.511
C06862=1051.432,146.272,-87.038,171.230,34.694,156.511
C06863=1051.438,146.521,-87.060,171.232,34.697,156.511
C06864=1051.444,146.770,-87.081,171.234,34.699,156.512
C06865=1051.450,147.019,-87.103,171.235,34.701,156.512
C06866=1051.456,147.268,-87.124,171.237,34.703,156.513
C06867=1051.462,147.517,-87.146,171.239,34.705,156.513
C06868=1051.468,147.766,-87.168,171.242,34.708,156.513
C06869=1051.474,148.015,-87.189,171.244,34.710,156.514
C06870=1051.479,148.264,-87.211,171.246,34.712,156.514
C06871=1051.486,148.513,-87.233,171.247,34.714,156.514
C06872=1051.492,148.762,-87.255,171.249,34.717,156.515
C06873=1051.498,149.011,-87.276,171.251,34.718,156.515
C06874=1051.504,149.260,-87.298,171.253,34.721,156.516
C06875=1051.510,149.509,-87.320,171.255,34.723,156.516
C06876=1051.516,149.758,-87.341,171.258,34.725,156.516
C06877=1051.523,150.007,-87.364,171.259,34.727,156.517
C06878=1051.527,150.256,-87.385,171.261,34.730,156.517
C06879=1051.534,150.505,-87.407,171.263,34.732,156.518
C06880=1051.540,150.754,-87.429,171.265,34.734,156.518
C06881=1051.546,151.003,-87.451,171.267,34.736,156.518
C06882=1051.552,151.252,-87.473,171.269,34.739,156.519
C06883=1051.557,151.501,-87.495,171.271,34.741,156.519
C06884=1051.563,151.750,-87.516,171.273,34.743,156.520
C06885=1051.570,151.998,-87.539,171.275,34.746,156.520
C06886=1051.576,152.248,-87.560,171.277,34.748,156.520
C06887=1051.582,152.497,-87.582,171.279,34.750,156.521
C06888=1051.587,152.745,-87.604,171.281,34.752,156.521
C06889=1051.593,152.994,-87.626,171.283,34.754,156.522
C06890=1051.600,153.243,-87.648,171.285,34.756,156.522
C06891=1051.606,153.492,-87.670,171.286,34.759,156.523
C06892=1051.612,153.742,-87.692,171.288,34.761,156.523
C06893=1051.618,153.991,-87.714,171.291,34.763,156.523
C06894=1051.624,154.239,-87.736,171.293,34.765,156.524
C06895=1051.630,154.488,-87.757,171.295,34.768,156.524
C06896=1051.636,154.737,-87.779,171.297,34.770,156.524
C06897=1051.642,154.986,-87.802,171.299,34.772,156.525
C06898=1051.648,155.235,-87.824,171.301,34.774,156.525
C06899=1051.654,155.484,-87.846,171.302,34.777,156.526
C06900=1051.660,155.733,-87.868,171.305,34.779,156.526
C06901=1051.666,155.983,-87.890,171.307,34.781,156.526
C06902=1051.672,156.231,-87.912,171.309,34.783,156.527
C06903=1051.677,156.480,-87.934,171.311,34.785,156.527
C06904=1051.684,156.728,-87.956,171.313,34.788,156.528
C06905=1051.689,156.978,-87.979,171.315,34.790,156.528
C06906=1051.696,157.227,-88.001,171.317,34.792,156.529
C06907=1051.702,157.476,-88.023,171.318,34.795,156.529
C06908=1051.709,157.760,-88.048,171.322,34.797,156.529
C06909=1051.716,158.046,-88.074,171.324,34.800,156.530
C06910=1051.723,158.330,-88.099,171.326,34.802,156.530
C06911=1051.729,158.616,-88.124,171.328,34.805,156.531
C06912=1051.735,158.864,-88.147,171.330,34.807,156.531
C06913=1051.741,159.114,-88.169,171.332,34.809,156.532
C06914=1051.747,159.363,-88.192,171.334,34.812,156.532
C06915=1051.753,159.612,-88.214,171.336,34.814,156.532
C06916=1051.759,159.860,-88.236,171.339,34.816,156.533
C06917=1051.765,160.110,-88.258,171.341,34.819,156.533
C06918=1051.771,160.358,-88.280,171.343,34.821,156.534
C06919=1051.777,160.607,-88.303,171.344,34.823,156.534
C06920=1051.783,160.857,-88.325,171.346,34.825,156.534
C06921=1051.789,161.105,-88.348,171.348,34.828,156.535
C06922=1051.795,161.354,-88.371,171.350,34.830,156.535
C06923=1051.801,161.604,-88.393,171.353,34.833,156.536
C06924=1051.807,161.852,-88.416,171.355,34.835,156.536
C06925=1051.812,162.101,-88.438,171.357,34.837,156.537
C06926=1051.817,162.350,-88.461,171.359,34.839,156.537
C06927=1051.824,162.599,-88.483,171.361,34.842,156.538
C06928=1051.829,162.848,-88.506,171.362,34.844,156.538
C06929=1051.835,163.097,-88.529,171.364,34.847,156.538
C06930=1051.841,163.345,-88.552,171.367,34.849,156.539
C06931=1051.847,163.595,-88.573,171.369,34.851,156.539
C06932=1051.853,163.844,-88.596,171.371,34.854,156.540
C06933=1051.858,164.092,-88.619,171.373,34.856,156.540
C06934=1051.864,164.341,-88.642,171.375,34.858,156.541
C06935=1051.870,164.590,-88.665,171.377,34.861,156.541
C06936=1051.876,164.839,-88.687,171.379,34.863,156.541
C06937=1051.882,165.088,-88.710,171.382,34.866,156.542
C06938=1051.888,165.337,-88.732,171.384,34.868,156.542
C06939=1051.893,165.586,-88.755,171.386,34.870,156.543
C06940=1051.900,165.835,-88.778,171.387,34.873,156.543
C06941=1051.905,166.084,-88.801,171.389,34.875,156.544
C06942=1051.911,166.333,-88.824,171.391,34.878,156.544
C06943=1051.917,166.581,-88.847,171.393,34.880,156.545
C06944=1051.923,166.830,-88.870,171.395,34.882,156.545
C06945=1051.929,167.080,-88.891,171.398,34.885,156.545
C06946=1051.935,167.328,-88.914,171.400,34.887,156.546
C06947=1051.940,167.577,-88.937,171.402,34.890,156.546
C06948=1051.946,167.826,-88.960,171.404,34.891,156.547
C06949=1051.952,168.075,-88.983,171.406,34.894,156.547
C06950=1051.958,168.324,-89.005,171.408,34.896,156.548
C06951=1051.964,168.573,-89.028,171.411,34.899,156.548
C06952=1051.970,168.821,-89.051,171.413,34.901,156.548
C06953=1051.975,169.070,-89.074,171.415,34.903,156.549
C06954=1051.981,169.319,-89.097,171.417,34.906,156.549
C06955=1051.988,169.568,-89.119,171.419,34.908,156.550
C06956=1051.993,169.817,-89.142,171.421,34.911,156.550
C06957=1051.999,170.066,-89.165,171.423,34.913,156.551
C06958=1052.005,170.315,-89.188,171.426,34.915,156.551
C06959=1052.011,170.563,-89.211,171.428,34.918,156.551
C06960=1052.017,170.813,-89.235,171.430,34.920,156.552
C06961=1052.024,171.061,-89.258,171.432,34.923,156.552
C06962=1052.029,171.310,-89.281,171.434,34.925,156.553
C06963=1052.035,171.559,-89.303,171.436,34.927,156.553
C06964=1052.041,171.808,-89.326,171.438,34.930,156.554
C06965=1052.047,172.057,-89.349,171.441,34.932,156.554
C06966=1052.052,172.305,-89.372,171.443,34.935,156.555
C06967=1052.059,172.554,-89.395,171.445,34.937,156.555
C06968=1052.065,172.804,-89.418,171.447,34.939,156.555
C06969=1052.071,173.053,-89.441,171.449,34.942,156.556
C06970=1052.077,173.301,-89.465,171.451,34.944,156.556
C06971=1052.083,173.550,-89.488,171.453,34.947,156.557
C06972=1052.089,173.834,-89.513,171.456,34.949,156.557
C06973=1052.097,174.119,-89.541,171.458,34.952,156.558
C06974=1052.103,174.404,-89.566,171.460,34.955,156.558
C06975=1052.110,174.688,-89.593,171.463,34.957,156.559
C06976=1052.116,174.937,-89.617,171.465,34.960,156.559
C06977=1052.123,175.186,-89.639,171.467,34.962,156.560
C06978=1052.128,175.435,-89.662,171.470,34.965,156.560
C06979=1052.134,175.684,-89.685,171.472,34.967,156.560
C06980=1052.141,175.933,-89.709,171.474,34.969,156.561
C06981=1052.146,176.182,-89.732,171.476,34.972,156.561
C06982=1052.152,176.430,-89.755,171.478,34.974,156.562
C06983=1052.158,176.679,-89.778,171.480,34.977,156.562
C06984=1052.164,176.928,-89.801,171.483,34.979,156.563
C06985=1052.170,177.177,-89.825,171.485,34.981,156.563
C06986=1052.177,177.426,-89.847,171.487,34.983,156.564
C06987=1052.183,177.674,-89.871,171.489,34.986,156.564
C06988=1052.189,177.924,-89.894,171.491,34.988,156.564
C06989=1052.195,178.173,-89.917,171.493,34.991,156.565
C06990=1052.201,178.421,-89.941,171.495,34.993,156.565
C06991=1052.207,178.670,-89.964,171.498,34.995,156.566
C06992=1052.213,178.919,-89.987,171.500,34.998,156.566
C06993=1052.219,179.168,-90.010,171.503,35.000,156.567
C06994=1052.225,179.416,-90.033,171.505,35.003,156.567
C06995=1052.231,179.665,-90.057,171.507,35.005,156.568
C06996=1052.238,179.914,-90.080,171.509,35.007,156.568
C06997=1052.244,180.162,-90.103,171.511,35.010,156.568
C06998=1052.250,180.412,-90.127,171.514,35.012,156.569
C06999=1052.256,180.661,-90.150,171.516,35.015,156.569
C07000=1052.262,180.909,-90.173,171.518,35.017,156.570
C07001=1052.268,181.159,-90.197,171.520,35.020,156.570
C07002=1052.274,181.407,-90.220,171.522,35.022,156.571
C07003=1052.280,181.656,-90.243,171.524,35.024,156.571
C07004=1052.287,181.905,-90.267,171.527,35.027,156.572
C07005=1052.292,182.154,-90.290,171.530,35.029,156.572
C07006=1052.298,182.402,-90.314,171.532,35.032,156.572
C07007=1052.305,182.652,-90.337,171.534,35.034,156.573
C07008=1052.311,182.900,-90.361,171.536,35.036,156.573
C07009=1052.317,183.149,-90.384,171.538,35.038,156.574
C07010=1052.324,183.397,-90.407,171.541,35.041,156.574
C07011=1052.330,183.646,-90.431,171.543,35.043,156.575
C07012=1052.336,183.895,-90.454,171.545,35.046,156.575
C07013=1052.342,184.144,-90.478,171.547,35.048,156.576
C07014=1052.348,184.394,-90.502,171.549,35.051,156.576
C07015=1052.354,184.642,-90.526,171.552,35.053,156.576
C07016=1052.359,184.890,-90.550,171.555,35.056,156.577
C07017=1052.366,185.139,-90.574,171.557,35.058,156.577
C07018=1052.371,185.389,-90.597,171.559,35.061,156.578
C07019=1052.377,185.637,-90.621,171.561,35.063,156.578
C07020=1052.383,185.885,-90.645,171.563,35.066,156.579
C07021=1052.389,186.134,-90.669,171.565,35.069,156.579
C07022=1052.395,186.383,-90.692,171.568,35.071,156.580
C07023=1052.400,186.632,-90.716,171.570,35.074,156.580
C07024=1052.407,186.881,-90.741,171.572,35.076,156.581
C07025=1052.412,187.129,-90.765,171.574,35.079,156.581
C07026=1052.419,187.378,-90.789,171.577,35.082,156.582
C07027=1052.423,187.628,-90.812,171.579,35.084,156.582
C07028=1052.430,187.876,-90.836,171.582,35.087,156.583
C07029=1052.435,188.125,-90.861,171.584,35.089,156.583
C07030=1052.441,188.373,-90.884,171.586,35.092,156.584
C07031=1052.447,188.622,-90.909,171.588,35.094,156.584
C07032=1052.453,188.871,-90.933,171.590,35.097,156.585
C07033=1052.459,189.119,-90.956,171.593,35.100,156.585
C07034=1052.465,189.369,-90.980,171.595,35.102,156.586
C07035=1052.471,189.618,-91.004,171.598,35.105,156.586
C07036=1052.477,189.901,-91.032,171.600,35.108,156.587
C07037=1052.484,190.186,-91.059,171.602,35.111,156.587
C07038=1052.491,190.470,-91.087,171.605,35.114,156.588
C07039=1052.498,190.755,-91.115,171.608,35.117,156.588
C07040=1052.504,191.003,-91.138,171.610,35.119,156.589
C07041=1052.510,191.252,-91.163,171.613,35.122,156.589
C07042=1052.516,191.500,-91.186,171.615,35.125,156.590
C07043=1052.521,191.749,-91.211,171.617,35.127,156.590
C07044=1052.528,191.998,-91.235,171.620,35.130,156.591
C07045=1052.533,192.247,-91.259,171.622,35.132,156.591
C07046=1052.540,192.496,-91.283,171.624,35.135,156.592
C07047=1052.545,192.744,-91.307,171.627,35.138,156.592
C07048=1052.552,192.993,-91.331,171.629,35.140,156.593
C07049=1052.557,193.242,-91.356,171.632,35.143,156.593
C07050=1052.564,193.491,-91.380,171.634,35.145,156.594
C07051=1052.569,193.739,-91.404,171.636,35.148,156.594
C07052=1052.576,193.988,-91.428,171.638,35.151,156.595
C07053=1052.581,194.237,-91.452,171.641,35.153,156.595
C07054=1052.587,194.485,-91.477,171.643,35.156,156.596
C07055=1052.594,194.734,-91.501,171.646,35.158,156.596
C07056=1052.599,194.983,-91.526,171.648,35.161,156.597
C07057=1052.606,195.232,-91.550,171.650,35.164,156.597
C07058=1052.611,195.481,-91.574,171.653,35.166,156.598
C07059=1052.618,195.730,-91.598,171.655,35.169,156.598
C07060=1052.623,195.978,-91.622,171.658,35.171,156.599
C07061=1052.630,196.227,-91.647,171.660,35.174,156.599
C07062=1052.636,196.476,-91.672,171.662,35.177,156.600
C07063=1052.642,196.724,-91.695,171.665,35.179,156.600
C07064=1052.648,196.973,-91.720,171.667,35.182,156.601
C07065=1052.653,197.221,-91.745,171.669,35.184,156.601
C07066=1052.660,197.470,-91.769,171.672,35.187,156.602
C07067=1052.666,197.720,-91.794,171.674,35.190,156.602
C07068=1052.672,197.968,-91.817,171.677,35.192,156.603
C07069=1052.678,198.217,-91.843,171.679,35.195,156.603
C07070=1052.684,198.465,-91.866,171.681,35.198,156.604
C07071=1052.690,198.714,-91.891,171.684,35.200,156.604
C07072=1052.696,198.963,-91.915,171.687,35.203,156.605
C07073=1052.702,199.211,-91.940,171.689,35.206,156.605
C07074=1052.708,199.460,-91.964,171.691,35.208,156.606
C07075=1052.715,199.709,-91.989,171.693,35.211,156.606
C07076=1052.720,199.957,-92.013,171.697,35.213,156.607
C07077=1052.727,200.206,-92.038,171.699,35.216,156.607
C07078=1052.733,200.455,-92.063,171.701,35.219,156.608
C07079=1052.739,200.704,-92.087,171.703,35.221,156.608
C07080=1052.745,200.953,-92.111,171.706,35.224,156.609
C07081=1052.751,201.201,-92.136,171.709,35.227,156.609
C07082=1052.758,201.450,-92.161,171.711,35.229,156.610
C07083=1052.764,201.698,-92.185,171.713,35.232,156.610
C07084=1052.770,201.947,-92.210,171.716,35.235,156.611
C07085=1052.776,202.196,-92.235,171.718,35.237,156.611
C07086=1052.781,202.445,-92.260,171.721,35.240,156.612
C07087=1052.787,202.693,-92.285,171.723,35.243,156.612
C07088=1052.793,202.943,-92.310,171.726,35.246,156.613
C07089=1052.800,203.190,-92.334,171.728,35.248,156.613
C07090=1052.805,203.440,-92.359,171.730,35.251,156.614
C07091=1052.812,203.688,-92.384,171.733,35.254,156.614
C07092=1052.817,203.937,-92.408,171.736,35.257,156.615
C07093=1052.823,204.186,-92.434,171.738,35.259,156.615
C07094=1052.829,204.434,-92.459,171.740,35.262,156.616
C07095=1052.835,204.683,-92.484,171.742,35.265,156.616
C07096=1052.841,204.931,-92.509,171.746,35.267,156.617
C07097=1052.847,205.181,-92.533,171.748,35.271,156.618
C07098=1052.853,205.429,-92.558,171.750,35.273,156.618
C07099=1052.859,205.678,-92.584,171.753,35.276,156.619
C07100=1052.884,206.730,-92.689,171.970,35.370,156.635
C07101=1052.892,206.974,-92.714,171.971,35.373,156.636
C07102=1052.897,207.219,-92.740,171.973,35.377,156.636
C07103=1052.904,207.465,-92.765,171.976,35.380,156.637
C07104=1052.910,207.710,-92.791,171.977,35.384,156.638
C07105=1052.916,207.955,-92.816,171.979,35.388,156.639
C07106=1052.923,208.200,-92.842,171.981,35.391,156.639
C07107=1052.929,208.445,-92.867,171.983,35.394,156.640
C07108=1052.935,208.690,-92.894,171.985,35.398,156.641
C07109=1052.941,208.939,-92.919,171.986,35.402,156.641
C07110=1052.948,209.188,-92.946,171.989,35.405,156.642
C07111=1052.954,209.436,-92.972,171.991,35.409,156.643
C07112=1052.960,209.685,-92.998,171.992,35.412,156.643
C07113=1052.966,209.933,-93.024,171.995,35.416,156.644
C07114=1052.973,210.182,-93.050,171.997,35.420,156.645
C07115=1052.979,210.431,-93.076,171.998,35.423,156.646
C07116=1052.985,210.679,-93.102,172.001,35.427,156.646
C07117=1052.993,210.927,-93.129,172.003,35.430,156.647
C07118=1052.998,211.176,-93.155,172.005,35.433,156.648
C07119=1053.005,211.424,-93.181,172.006,35.437,156.648
C07120=1053.012,211.673,-93.207,172.009,35.441,156.649
C07121=1053.017,211.922,-93.234,172.011,35.444,156.650
C07122=1053.024,212.170,-93.259,172.012,35.448,156.651
C07123=1053.030,212.419,-93.286,172.015,35.452,156.651
C07124=1053.037,212.667,-93.312,172.017,35.455,156.652
C07125=1053.042,212.916,-93.339,172.018,35.459,156.653
C07126=1053.049,213.164,-93.365,172.021,35.462,156.653
C07127=1053.055,213.413,-93.392,172.023,35.466,156.654
C07128=1053.061,213.662,-93.417,172.025,35.470,156.655
C07129=1053.068,213.911,-93.444,172.027,35.473,156.656
C07130=1053.074,214.159,-93.470,172.029,35.477,156.656
C07131=1053.080,214.407,-93.497,172.031,35.480,156.657
C07132=1053.087,214.656,-93.523,172.033,35.484,156.658
C07133=1053.093,214.904,-93.550,172.035,35.487,156.658
C07134=1053.099,215.152,-93.577,172.037,35.491,156.659
C07135=1053.106,215.401,-93.603,172.039,35.494,156.660
C07136=1053.112,215.650,-93.630,172.041,35.498,156.661
C07137=1053.118,215.898,-93.655,172.043,35.501,156.661
C07138=1053.124,216.147,-93.682,172.045,35.505,156.662
C07139=1053.131,216.395,-93.708,172.048,35.509,156.663
C07140=1053.137,216.644,-93.735,172.049,35.512,156.664
C07141=1053.144,216.892,-93.761,172.051,35.516,156.664
C07142=1053.149,217.141,-93.788,172.054,35.519,156.665
C07143=1053.156,217.390,-93.815,172.056,35.523,156.666
C07144=1053.162,217.638,-93.841,172.057,35.526,156.666
C07145=1053.169,217.887,-93.868,172.060,35.530,156.667
C07146=1053.175,218.135,-93.894,172.062,35.533,156.668
C07147=1053.181,218.384,-93.921,172.064,35.537,156.668
C07148=1053.188,218.632,-93.948,172.067,35.541,156.669
C07149=1053.194,218.880,-93.974,172.068,35.544,156.670
C07150=1053.200,219.129,-94.001,172.070,35.547,156.671
C07151=1053.207,219.377,-94.028,172.073,35.551,156.671
C07152=1053.213,219.626,-94.055,172.075,35.554,156.672
C07153=1053.220,219.874,-94.081,172.076,35.558,156.673
C07154=1053.226,220.123,-94.108,172.078,35.561,156.673
C07155=1053.232,220.372,-94.134,172.081,35.565,156.674
C07156=1053.239,220.620,-94.161,172.083,35.568,156.675
C07157=1053.245,220.868,-94.188,172.085,35.572,156.676
C07158=1053.252,221.116,-94.214,172.087,35.575,156.676
C07159=1053.258,221.364,-94.241,172.089,35.579,156.677
C07160=1053.265,221.611,-94.268,172.091,35.583,156.678
C07161=1053.270,221.860,-94.295,172.094,35.586,156.678
C07162=1053.277,222.106,-94.321,172.096,35.589,156.679
C07163=1053.283,222.354,-94.349,172.097,35.593,156.680
C07164=1053.288,222.602,-94.375,172.100,35.596,156.680
C07165=1053.296,222.851,-94.402,172.102,35.600,156.681
C07166=1053.302,223.099,-94.429,172.104,35.604,156.682
C07167=1053.308,223.348,-94.456,172.107,35.607,156.683
C07168=1053.314,223.596,-94.483,172.108,35.610,156.683
C07169=1053.320,223.845,-94.510,172.110,35.614,156.684
C07170=1053.326,224.093,-94.537,172.113,35.617,156.685
C07171=1053.333,224.342,-94.564,172.115,35.621,156.685
C07172=1053.339,224.590,-94.591,172.117,35.625,156.686
C07173=1053.346,224.839,-94.618,172.120,35.628,156.687
C07174=1053.352,225.088,-94.645,172.121,35.632,156.688
C07175=1053.358,225.335,-94.672,172.123,35.635,156.688
C07176=1053.365,225.584,-94.699,172.126,35.638,156.689
C07177=1053.371,225.832,-94.727,172.128,35.642,156.690
C07178=1053.378,226.081,-94.753,172.130,35.646,156.690
C07179=1053.384,226.329,-94.780,172.133,35.649,156.691
C07180=1053.390,226.578,-94.807,172.134,35.652,156.692
C07181=1053.397,226.827,-94.835,172.136,35.656,156.693
C07182=1053.403,227.075,-94.862,172.139,35.659,156.693
C07183=1053.409,227.324,-94.889,172.141,35.663,156.694
C07184=1053.415,227.571,-94.916,172.143,35.667,156.695
C07185=1053.422,227.820,-94.943,172.145,35.670,156.695
C07186=1053.428,228.069,-94.971,172.148,35.673,156.696
C07187=1053.435,228.317,-94.997,172.150,35.677,156.697
C07188=1053.441,228.565,-95.025,172.152,35.680,156.698
C07189=1053.448,228.814,-95.052,172.154,35.683,156.698
C07190=1053.454,229.062,-95.079,172.156,35.687,156.699
C07191=1053.460,229.311,-95.106,172.158,35.690,156.700
C07192=1053.467,229.560,-95.134,172.161,35.694,156.700
C07193=1053.473,229.807,-95.161,172.163,35.698,156.701
C07194=1053.479,230.056,-95.188,172.165,35.701,156.702
C07195=1053.486,230.304,-95.216,172.168,35.704,156.702
C07196=1053.491,230.553,-95.244,172.170,35.708,156.703
C07197=1053.498,230.802,-95.271,172.172,35.711,156.704
C07198=1053.504,231.050,-95.298,172.174,35.715,156.705
C07199=1053.511,231.298,-95.326,172.176,35.719,156.705
C07200=1053.517,231.547,-95.353,172.178,35.722,156.706
C07201=1053.523,231.795,-95.380,172.181,35.725,156.707
C07202=1053.530,232.043,-95.408,172.183,35.729,156.707
C07203=1053.536,232.292,-95.435,172.186,35.732,156.708
C07204=1053.542,232.540,-95.463,172.188,35.736,156.709
C07205=1053.548,232.789,-95.491,172.190,35.739,156.709
C07206=1053.555,233.037,-95.519,172.193,35.743,156.710
C07207=1053.561,233.286,-95.545,172.195,35.746,156.711
C07208=1053.567,233.534,-95.573,172.196,35.750,156.712
C07209=1053.574,233.783,-95.601,172.199,35.753,156.712
C07210=1053.579,234.031,-95.629,172.201,35.757,156.713
C07211=1053.586,234.279,-95.656,172.203,35.760,156.714
C07212=1053.593,234.528,-95.684,172.206,35.763,156.714
C07213=1053.598,234.772,-95.711,172.208,35.767,156.715
C07214=1053.605,235.015,-95.738,172.210,35.771,156.716
C07215=1053.611,235.260,-95.765,172.213,35.774,156.717
C07216=1053.617,235.503,-95.793,172.215,35.777,156.717
C07217=1053.623,235.747,-95.820,172.217,35.781,156.718
C07218=1053.629,235.992,-95.847,172.220,35.784,156.719
C07219=1053.635,236.235,-95.875,172.222,35.787,156.719
C07220=1053.642,236.479,-95.901,172.223,35.791,156.720
C07221=1053.648,236.728,-95.930,172.226,35.795,156.721
C07222=1053.654,236.976,-95.957,172.228,35.798,156.721
C07223=1053.661,237.225,-95.985,172.230,35.801,156.722
C07224=1053.667,237.472,-96.012,172.233,35.805,156.723
C07225=1053.673,237.721,-96.041,172.235,35.808,156.724
C07226=1053.680,237.970,-96.069,172.237,35.811,156.724
C07227=1053.686,238.218,-96.096,172.240,35.815,156.725
C07228=1053.693,238.466,-96.124,172.242,35.818,156.726
C07229=1053.699,238.715,-96.152,172.244,35.822,156.726
C07230=1053.705,238.963,-96.180,172.247,35.825,156.727
C07231=1053.712,239.211,-96.207,172.249,35.829,156.728
C07232=1053.718,239.460,-96.236,172.251,35.832,156.729
C07233=1053.725,239.709,-96.263,172.254,35.836,156.729
C07234=1053.731,239.956,-96.291,172.256,35.839,156.730
C07235=1053.737,240.205,-96.319,172.258,35.842,156.731
C07236=1053.744,240.453,-96.348,172.261,35.846,156.731
C07237=1053.749,240.702,-96.376,172.263,35.849,156.732
C07238=1053.756,240.950,-96.404,172.266,35.853,156.733
C07239=1053.763,241.199,-96.431,172.268,35.856,156.733
C07240=1053.769,241.447,-96.460,172.270,35.860,156.734
C07241=1053.775,241.696,-96.487,172.273,35.863,156.735
C07242=1053.782,241.943,-96.516,172.275,35.867,156.736
C07243=1053.788,242.192,-96.544,172.277,35.870,156.736
C07244=1053.794,242.440,-96.572,172.280,35.873,156.737
C07245=1053.800,242.689,-96.600,172.282,35.877,156.738
C07246=1053.807,242.937,-96.629,172.284,35.880,156.739
C07247=1053.813,243.185,-96.657,172.287,35.884,156.739
C07248=1053.819,243.433,-96.685,172.289,35.888,156.740
C07249=1053.825,243.682,-96.714,172.291,35.891,156.741
C07250=1053.832,243.930,-96.741,172.294,35.894,156.741
C07251=1053.838,244.179,-96.770,172.297,35.898,156.742
C07252=1053.845,244.427,-96.798,172.300,35.901,156.743
C07253=1053.850,244.675,-96.826,172.302,35.905,156.744
C07254=1053.857,244.924,-96.854,172.304,35.908,156.744
C07255=1053.863,245.172,-96.883,172.307,35.911,156.745
C07256=1053.869,245.421,-96.912,172.309,35.915,156.746
C07257=1053.876,245.669,-96.939,172.311,35.919,156.746
C07258=1053.882,245.917,-96.968,172.314,35.922,156.747
C07259=1053.888,246.165,-96.996,172.316,35.925,156.748
C07260=1053.895,246.413,-97.025,172.318,35.929,156.748
C07261=1053.901,246.662,-97.053,172.321,35.932,156.749
C07262=1053.907,246.910,-97.082,172.323,35.936,156.750
C07263=1053.913,247.159,-97.110,172.326,35.939,156.751
